//     PlcTask Inputs/GVL_iXlinker.EtherCAT_Master_ERxxxx.Beckhoff_ER3xxx.Beckhoff_ER3xxxEK1122.A_0012_ER3314_0002_0021.TC_Inputs_Channel_1.Status/Underrange <-> TC Inputs Channel 1/Status/Underrange
//     PlcTask Inputs/GVL_iXlinker.EtherCAT_Master_ERxxxx.Beckhoff_ER3xxx.Beckhoff_ER3xxxEK1122.A_0012_ER3314_0002_0021.TC_Inputs_Channel_2.Status/Underrange <-> TC Inputs Channel 2/Status/Underrange
//     PlcTask Inputs/GVL_iXlinker.EtherCAT_Master_ERxxxx.Beckhoff_ER3xxx.Beckhoff_ER3xxxEK1122.A_0012_ER3314_0002_0021.TC_Inputs_Channel_3.Status/Underrange <-> TC Inputs Channel 3/Status/Underrange
//     PlcTask Inputs/GVL_iXlinker.EtherCAT_Master_ERxxxx.Beckhoff_ER3xxx.Beckhoff_ER3xxxEK1122.A_0012_ER3314_0002_0021.TC_Inputs_Channel_4.Status/Underrange <-> TC Inputs Channel 4/Status/Underrange
//     PlcTask Inputs/GVL_iXlinker.EtherCAT_Master_ERxxxx.Beckhoff_ER3xxx.Beckhoff_ER3xxxEK1122.A_0012_ER3314_0002_0021.TC_Inputs_Channel_1.Status/Overrange <-> TC Inputs Channel 1/Status/Overrange
//     PlcTask Inputs/GVL_iXlinker.EtherCAT_Master_ERxxxx.Beckhoff_ER3xxx.Beckhoff_ER3xxxEK1122.A_0012_ER3314_0002_0021.TC_Inputs_Channel_2.Status/Overrange <-> TC Inputs Channel 2/Status/Overrange
//     PlcTask Inputs/GVL_iXlinker.EtherCAT_Master_ERxxxx.Beckhoff_ER3xxx.Beckhoff_ER3xxxEK1122.A_0012_ER3314_0002_0021.TC_Inputs_Channel_3.Status/Overrange <-> TC Inputs Channel 3/Status/Overrange
//     PlcTask Inputs/GVL_iXlinker.EtherCAT_Master_ERxxxx.Beckhoff_ER3xxx.Beckhoff_ER3xxxEK1122.A_0012_ER3314_0002_0021.TC_Inputs_Channel_4.Status/Overrange <-> TC Inputs Channel 4/Status/Overrange
//     PlcTask Inputs/GVL_iXlinker.EtherCAT_Master_ERxxxx.Beckhoff_ER3xxx.Beckhoff_ER3xxxEK1122.A_0012_ER3314_0002_0021.TC_Inputs_Channel_1.Status/Limit_1 <-> TC Inputs Channel 1/Status/Limit 1
//     PlcTask Inputs/GVL_iXlinker.EtherCAT_Master_ERxxxx.Beckhoff_ER3xxx.Beckhoff_ER3xxxEK1122.A_0012_ER3314_0002_0021.TC_Inputs_Channel_1.Status/Limit_2 <-> TC Inputs Channel 1/Status/Limit 2
//     PlcTask Inputs/GVL_iXlinker.EtherCAT_Master_ERxxxx.Beckhoff_ER3xxx.Beckhoff_ER3xxxEK1122.A_0012_ER3314_0002_0021.TC_Inputs_Channel_2.Status/Limit_1 <-> TC Inputs Channel 2/Status/Limit 1
//     PlcTask Inputs/GVL_iXlinker.EtherCAT_Master_ERxxxx.Beckhoff_ER3xxx.Beckhoff_ER3xxxEK1122.A_0012_ER3314_0002_0021.TC_Inputs_Channel_2.Status/Limit_2 <-> TC Inputs Channel 2/Status/Limit 2
//     PlcTask Inputs/GVL_iXlinker.EtherCAT_Master_ERxxxx.Beckhoff_ER3xxx.Beckhoff_ER3xxxEK1122.A_0012_ER3314_0002_0021.TC_Inputs_Channel_3.Status/Limit_1 <-> TC Inputs Channel 3/Status/Limit 1
//     PlcTask Inputs/GVL_iXlinker.EtherCAT_Master_ERxxxx.Beckhoff_ER3xxx.Beckhoff_ER3xxxEK1122.A_0012_ER3314_0002_0021.TC_Inputs_Channel_3.Status/Limit_2 <-> TC Inputs Channel 3/Status/Limit 2
//     PlcTask Inputs/GVL_iXlinker.EtherCAT_Master_ERxxxx.Beckhoff_ER3xxx.Beckhoff_ER3xxxEK1122.A_0012_ER3314_0002_0021.TC_Inputs_Channel_4.Status/Limit_1 <-> TC Inputs Channel 4/Status/Limit 1
//     PlcTask Inputs/GVL_iXlinker.EtherCAT_Master_ERxxxx.Beckhoff_ER3xxx.Beckhoff_ER3xxxEK1122.A_0012_ER3314_0002_0021.TC_Inputs_Channel_4.Status/Limit_2 <-> TC Inputs Channel 4/Status/Limit 2
//     PlcTask Inputs/GVL_iXlinker.EtherCAT_Master_ERxxxx.Beckhoff_ER3xxx.Beckhoff_ER3xxxEK1122.A_0012_ER3314_0002_0021.TC_Inputs_Channel_1.Status/Error <-> TC Inputs Channel 1/Status/Error
//     PlcTask Inputs/GVL_iXlinker.EtherCAT_Master_ERxxxx.Beckhoff_ER3xxx.Beckhoff_ER3xxxEK1122.A_0012_ER3314_0002_0021.TC_Inputs_Channel_2.Status/Error <-> TC Inputs Channel 2/Status/Error
//     PlcTask Inputs/GVL_iXlinker.EtherCAT_Master_ERxxxx.Beckhoff_ER3xxx.Beckhoff_ER3xxxEK1122.A_0012_ER3314_0002_0021.TC_Inputs_Channel_3.Status/Error <-> TC Inputs Channel 3/Status/Error
//     PlcTask Inputs/GVL_iXlinker.EtherCAT_Master_ERxxxx.Beckhoff_ER3xxx.Beckhoff_ER3xxxEK1122.A_0012_ER3314_0002_0021.TC_Inputs_Channel_4.Status/Error <-> TC Inputs Channel 4/Status/Error
//     PlcTask Inputs/GVL_iXlinker.EtherCAT_Master_ERxxxx.Beckhoff_ER3xxx.Beckhoff_ER3xxxEK1122.A_0012_ER3314_0002_0021.TC_Inputs_Channel_1.Status/TxPDO_State <-> TC Inputs Channel 1/Status/TxPDO State
//     PlcTask Inputs/GVL_iXlinker.EtherCAT_Master_ERxxxx.Beckhoff_ER3xxx.Beckhoff_ER3xxxEK1122.A_0012_ER3314_0002_0021.TC_Inputs_Channel_2.Status/TxPDO_State <-> TC Inputs Channel 2/Status/TxPDO State
//     PlcTask Inputs/GVL_iXlinker.EtherCAT_Master_ERxxxx.Beckhoff_ER3xxx.Beckhoff_ER3xxxEK1122.A_0012_ER3314_0002_0021.TC_Inputs_Channel_3.Status/TxPDO_State <-> TC Inputs Channel 3/Status/TxPDO State
//     PlcTask Inputs/GVL_iXlinker.EtherCAT_Master_ERxxxx.Beckhoff_ER3xxx.Beckhoff_ER3xxxEK1122.A_0012_ER3314_0002_0021.TC_Inputs_Channel_4.Status/TxPDO_State <-> TC Inputs Channel 4/Status/TxPDO State
//     PlcTask Inputs/GVL_iXlinker.EtherCAT_Master_ERxxxx.Beckhoff_ER3xxx.Beckhoff_ER3xxxEK1122.A_0012_ER3314_0002_0021.TC_Inputs_Channel_1.Status/TxPDO_Toggle <-> TC Inputs Channel 1/Status/TxPDO Toggle
//     PlcTask Inputs/GVL_iXlinker.EtherCAT_Master_ERxxxx.Beckhoff_ER3xxx.Beckhoff_ER3xxxEK1122.A_0012_ER3314_0002_0021.TC_Inputs_Channel_2.Status/TxPDO_Toggle <-> TC Inputs Channel 2/Status/TxPDO Toggle
//     PlcTask Inputs/GVL_iXlinker.EtherCAT_Master_ERxxxx.Beckhoff_ER3xxx.Beckhoff_ER3xxxEK1122.A_0012_ER3314_0002_0021.TC_Inputs_Channel_3.Status/TxPDO_Toggle <-> TC Inputs Channel 3/Status/TxPDO Toggle
//     PlcTask Inputs/GVL_iXlinker.EtherCAT_Master_ERxxxx.Beckhoff_ER3xxx.Beckhoff_ER3xxxEK1122.A_0012_ER3314_0002_0021.TC_Inputs_Channel_4.Status/TxPDO_Toggle <-> TC Inputs Channel 4/Status/TxPDO Toggle
//     PlcTask Inputs/GVL_iXlinker.EtherCAT_Master_ERxxxx.Beckhoff_ER3xxx.Beckhoff_ER3xxxEK1122.A_0012_ER3314_0002_0021.TC_Inputs_Channel_1.Value <-> TC Inputs Channel 1/Value
//     PlcTask Inputs/GVL_iXlinker.EtherCAT_Master_ERxxxx.Beckhoff_ER3xxx.Beckhoff_ER3xxxEK1122.A_0012_ER3314_0002_0021.TC_Inputs_Channel_2.Value <-> TC Inputs Channel 2/Value
//     PlcTask Inputs/GVL_iXlinker.EtherCAT_Master_ERxxxx.Beckhoff_ER3xxx.Beckhoff_ER3xxxEK1122.A_0012_ER3314_0002_0021.TC_Inputs_Channel_3.Value <-> TC Inputs Channel 3/Value
//     PlcTask Inputs/GVL_iXlinker.EtherCAT_Master_ERxxxx.Beckhoff_ER3xxx.Beckhoff_ER3xxxEK1122.A_0012_ER3314_0002_0021.TC_Inputs_Channel_4.Value <-> TC Inputs Channel 4/Value
//     PlcTask Inputs/GVL_iXlinker.EtherCAT_Master_ERxxxx.Beckhoff_ER3xxx.Beckhoff_ER3xxxEK1122.A_0012_ER3314_0002_0021.WcState.WcState <-> WcState/WcState
//     PlcTask Inputs/GVL_iXlinker.EtherCAT_Master_ERxxxx.Beckhoff_ER3xxx.Beckhoff_ER3xxxEK1122.A_0012_ER3314_0002_0021.WcState.InputToggle <-> WcState/InputToggle
//     PlcTask Inputs/GVL_iXlinker.EtherCAT_Master_ERxxxx.Beckhoff_ER3xxx.Beckhoff_ER3xxxEK1122.A_0012_ER3314_0002_0021.InfoData.AdsAddr <-> InfoData/AdsAddr
//     PlcTask Inputs/GVL_iXlinker.EtherCAT_Master_ERxxxx.Beckhoff_ER3xxx.Beckhoff_ER3xxxEK1122.A_0012_ER3314_0002_0021.InfoData.State <-> InfoData/State
//   PLC/PLC Instance <-> EtherCAT Master ERxxxx/Beckhoff ER4xxx
//     PlcTask Inputs/GVL_iXlinker.EtherCAT_Master_ERxxxx.Beckhoff_ER4xxx.InfoData.State <-> InfoData/State
//   PLC/PLC Instance <-> EtherCAT Master ERxxxx/Beckhoff ER4xxx/Beckhoff ER4xxxEK1122
//     PlcTask Inputs/GVL_iXlinker.EtherCAT_Master_ERxxxx.Beckhoff_ER4xxx.Beckhoff_ER4xxxEK1122.InfoData.State <-> InfoData/State
//   PLC/PLC Instance <-> EtherCAT Master ERxxxx/Beckhoff ER4xxx/Beckhoff ER4xxxEK1122/Beckhoff ER4xxxsub EK1100
//     PlcTask Inputs/GVL_iXlinker.EtherCAT_Master_ERxxxx.Beckhoff_ER4xxx.Beckhoff_ER4xxxEK1122.Beckhoff_ER4xxxsub_EK1100.InfoData.State <-> InfoData/State
//   PLC/PLC Instance <-> EtherCAT Master ERxxxx/Beckhoff ER4xxx/Beckhoff ER4xxxEK1122/A_0001(ER4174-0002-0016)
//     PlcTask Outputs/GVL_iXlinker.EtherCAT_Master_ERxxxx.Beckhoff_ER4xxx.Beckhoff_ER4xxxEK1122.A_0001_ER4174_0002_0016.AO_Outputs_Channel_1.Analog_output <-> AO Outputs Channel 1/Analog output
//     PlcTask Outputs/GVL_iXlinker.EtherCAT_Master_ERxxxx.Beckhoff_ER4xxx.Beckhoff_ER4xxxEK1122.A_0001_ER4174_0002_0016.AO_Outputs_Channel_2.Analog_output <-> AO Outputs Channel 2/Analog output
//     PlcTask Outputs/GVL_iXlinker.EtherCAT_Master_ERxxxx.Beckhoff_ER4xxx.Beckhoff_ER4xxxEK1122.A_0001_ER4174_0002_0016.AO_Outputs_Channel_3.Analog_output <-> AO Outputs Channel 3/Analog output
//     PlcTask Outputs/GVL_iXlinker.EtherCAT_Master_ERxxxx.Beckhoff_ER4xxx.Beckhoff_ER4xxxEK1122.A_0001_ER4174_0002_0016.AO_Outputs_Channel_4.Analog_output <-> AO Outputs Channel 4/Analog output
//     PlcTask Inputs/GVL_iXlinker.EtherCAT_Master_ERxxxx.Beckhoff_ER4xxx.Beckhoff_ER4xxxEK1122.A_0001_ER4174_0002_0016.WcState.WcState <-> WcState/WcState
//     PlcTask Inputs/GVL_iXlinker.EtherCAT_Master_ERxxxx.Beckhoff_ER4xxx.Beckhoff_ER4xxxEK1122.A_0001_ER4174_0002_0016.InfoData.AdsAddr <-> InfoData/AdsAddr
//     PlcTask Inputs/GVL_iXlinker.EtherCAT_Master_ERxxxx.Beckhoff_ER4xxx.Beckhoff_ER4xxxEK1122.A_0001_ER4174_0002_0016.InfoData.State <-> InfoData/State
//   PLC/PLC Instance <-> EtherCAT Master ERxxxx/Beckhoff ER4xxx/Beckhoff ER4xxxEK1122/A_0002(ER4174-0002-0019)
//     PlcTask Outputs/GVL_iXlinker.EtherCAT_Master_ERxxxx.Beckhoff_ER4xxx.Beckhoff_ER4xxxEK1122.A_0002_ER4174_0002_0019.AO_Outputs_Channel_1.Analog_output <-> AO Outputs Channel 1/Analog output
//     PlcTask Outputs/GVL_iXlinker.EtherCAT_Master_ERxxxx.Beckhoff_ER4xxx.Beckhoff_ER4xxxEK1122.A_0002_ER4174_0002_0019.AO_Outputs_Channel_2.Analog_output <-> AO Outputs Channel 2/Analog output
//     PlcTask Outputs/GVL_iXlinker.EtherCAT_Master_ERxxxx.Beckhoff_ER4xxx.Beckhoff_ER4xxxEK1122.A_0002_ER4174_0002_0019.AO_Outputs_Channel_3.Analog_output <-> AO Outputs Channel 3/Analog output
//     PlcTask Outputs/GVL_iXlinker.EtherCAT_Master_ERxxxx.Beckhoff_ER4xxx.Beckhoff_ER4xxxEK1122.A_0002_ER4174_0002_0019.AO_Outputs_Channel_4.Analog_output <-> AO Outputs Channel 4/Analog output
//     PlcTask Inputs/GVL_iXlinker.EtherCAT_Master_ERxxxx.Beckhoff_ER4xxx.Beckhoff_ER4xxxEK1122.A_0002_ER4174_0002_0019.WcState.WcState <-> WcState/WcState
//     PlcTask Inputs/GVL_iXlinker.EtherCAT_Master_ERxxxx.Beckhoff_ER4xxx.Beckhoff_ER4xxxEK1122.A_0002_ER4174_0002_0019.InfoData.AdsAddr <-> InfoData/AdsAddr
//     PlcTask Inputs/GVL_iXlinker.EtherCAT_Master_ERxxxx.Beckhoff_ER4xxx.Beckhoff_ER4xxxEK1122.A_0002_ER4174_0002_0019.InfoData.State <-> InfoData/State
//   PLC/PLC Instance <-> EtherCAT Master ERxxxx/Beckhoff ER4xxx/Beckhoff ER4xxxEK1122/A_0003(ER4374-0002-0018)
//     PlcTask Inputs/GVL_iXlinker.EtherCAT_Master_ERxxxx.Beckhoff_ER4xxx.Beckhoff_ER4xxxEK1122.A_0003_ER4374_0002_0018.AI_Inputs_Channel_1.Status/Underrange <-> AI Inputs Channel 1/Status/Underrange
//     PlcTask Inputs/GVL_iXlinker.EtherCAT_Master_ERxxxx.Beckhoff_ER4xxx.Beckhoff_ER4xxxEK1122.A_0003_ER4374_0002_0018.AI_Inputs_Channel_2.Status/Underrange <-> AI Inputs Channel 2/Status/Underrange
//     PlcTask Inputs/GVL_iXlinker.EtherCAT_Master_ERxxxx.Beckhoff_ER4xxx.Beckhoff_ER4xxxEK1122.A_0003_ER4374_0002_0018.AI_Inputs_Channel_1.Status/Overrange <-> AI Inputs Channel 1/Status/Overrange
//     PlcTask Inputs/GVL_iXlinker.EtherCAT_Master_ERxxxx.Beckhoff_ER4xxx.Beckhoff_ER4xxxEK1122.A_0003_ER4374_0002_0018.AI_Inputs_Channel_2.Status/Overrange <-> AI Inputs Channel 2/Status/Overrange
//     PlcTask Inputs/GVL_iXlinker.EtherCAT_Master_ERxxxx.Beckhoff_ER4xxx.Beckhoff_ER4xxxEK1122.A_0003_ER4374_0002_0018.AI_Inputs_Channel_1.Status/Limit_1 <-> AI Inputs Channel 1/Status/Limit 1
//     PlcTask Inputs/GVL_iXlinker.EtherCAT_Master_ERxxxx.Beckhoff_ER4xxx.Beckhoff_ER4xxxEK1122.A_0003_ER4374_0002_0018.AI_Inputs_Channel_1.Status/Limit_2 <-> AI Inputs Channel 1/Status/Limit 2
//     PlcTask Inputs/GVL_iXlinker.EtherCAT_Master_ERxxxx.Beckhoff_ER4xxx.Beckhoff_ER4xxxEK1122.A_0003_ER4374_0002_0018.AI_Inputs_Channel_2.Status/Limit_1 <-> AI Inputs Channel 2/Status/Limit 1
//     PlcTask Inputs/GVL_iXlinker.EtherCAT_Master_ERxxxx.Beckhoff_ER4xxx.Beckhoff_ER4xxxEK1122.A_0003_ER4374_0002_0018.AI_Inputs_Channel_2.Status/Limit_2 <-> AI Inputs Channel 2/Status/Limit 2
//     PlcTask Inputs/GVL_iXlinker.EtherCAT_Master_ERxxxx.Beckhoff_ER4xxx.Beckhoff_ER4xxxEK1122.A_0003_ER4374_0002_0018.AI_Inputs_Channel_1.Status/Error <-> AI Inputs Channel 1/Status/Error
//     PlcTask Inputs/GVL_iXlinker.EtherCAT_Master_ERxxxx.Beckhoff_ER4xxx.Beckhoff_ER4xxxEK1122.A_0003_ER4374_0002_0018.AI_Inputs_Channel_2.Status/Error <-> AI Inputs Channel 2/Status/Error
//     PlcTask Inputs/GVL_iXlinker.EtherCAT_Master_ERxxxx.Beckhoff_ER4xxx.Beckhoff_ER4xxxEK1122.A_0003_ER4374_0002_0018.AI_Inputs_Channel_1.Status/Sync_error <-> AI Inputs Channel 1/Status/Sync error
//     PlcTask Inputs/GVL_iXlinker.EtherCAT_Master_ERxxxx.Beckhoff_ER4xxx.Beckhoff_ER4xxxEK1122.A_0003_ER4374_0002_0018.AI_Inputs_Channel_2.Status/Sync_error <-> AI Inputs Channel 2/Status/Sync error
//     PlcTask Inputs/GVL_iXlinker.EtherCAT_Master_ERxxxx.Beckhoff_ER4xxx.Beckhoff_ER4xxxEK1122.A_0003_ER4374_0002_0018.AI_Inputs_Channel_1.Status/TxPDO_State <-> AI Inputs Channel 1/Status/TxPDO State
//     PlcTask Inputs/GVL_iXlinker.EtherCAT_Master_ERxxxx.Beckhoff_ER4xxx.Beckhoff_ER4xxxEK1122.A_0003_ER4374_0002_0018.AI_Inputs_Channel_2.Status/TxPDO_State <-> AI Inputs Channel 2/Status/TxPDO State
//     PlcTask Inputs/GVL_iXlinker.EtherCAT_Master_ERxxxx.Beckhoff_ER4xxx.Beckhoff_ER4xxxEK1122.A_0003_ER4374_0002_0018.AI_Inputs_Channel_1.Status/TxPDO_Toggle <-> AI Inputs Channel 1/Status/TxPDO Toggle
//     PlcTask Inputs/GVL_iXlinker.EtherCAT_Master_ERxxxx.Beckhoff_ER4xxx.Beckhoff_ER4xxxEK1122.A_0003_ER4374_0002_0018.AI_Inputs_Channel_2.Status/TxPDO_Toggle <-> AI Inputs Channel 2/Status/TxPDO Toggle
//     PlcTask Inputs/GVL_iXlinker.EtherCAT_Master_ERxxxx.Beckhoff_ER4xxx.Beckhoff_ER4xxxEK1122.A_0003_ER4374_0002_0018.AI_Inputs_Channel_1.Value <-> AI Inputs Channel 1/Value
//     PlcTask Inputs/GVL_iXlinker.EtherCAT_Master_ERxxxx.Beckhoff_ER4xxx.Beckhoff_ER4xxxEK1122.A_0003_ER4374_0002_0018.AI_Inputs_Channel_2.Value <-> AI Inputs Channel 2/Value
//     PlcTask Outputs/GVL_iXlinker.EtherCAT_Master_ERxxxx.Beckhoff_ER4xxx.Beckhoff_ER4xxxEK1122.A_0003_ER4374_0002_0018.AO_Outputs_Channel_3.Analog_output <-> AO Outputs Channel 3/Analog output
//     PlcTask Outputs/GVL_iXlinker.EtherCAT_Master_ERxxxx.Beckhoff_ER4xxx.Beckhoff_ER4xxxEK1122.A_0003_ER4374_0002_0018.AO_Outputs_Channel_4.Analog_output <-> AO Outputs Channel 4/Analog output
//     PlcTask Inputs/GVL_iXlinker.EtherCAT_Master_ERxxxx.Beckhoff_ER4xxx.Beckhoff_ER4xxxEK1122.A_0003_ER4374_0002_0018.WcState.WcState <-> WcState/WcState
//     PlcTask Inputs/GVL_iXlinker.EtherCAT_Master_ERxxxx.Beckhoff_ER4xxx.Beckhoff_ER4xxxEK1122.A_0003_ER4374_0002_0018.WcState.InputToggle <-> WcState/InputToggle
//     PlcTask Inputs/GVL_iXlinker.EtherCAT_Master_ERxxxx.Beckhoff_ER4xxx.Beckhoff_ER4xxxEK1122.A_0003_ER4374_0002_0018.InfoData.AdsAddr <-> InfoData/AdsAddr
//     PlcTask Inputs/GVL_iXlinker.EtherCAT_Master_ERxxxx.Beckhoff_ER4xxx.Beckhoff_ER4xxxEK1122.A_0003_ER4374_0002_0018.InfoData.State <-> InfoData/State
//   PLC/PLC Instance <-> EtherCAT Master ERxxxx/Beckhoff ER4xxx/Beckhoff ER4xxxEK1122/A_0004(ER4374-0002-0019)
//     PlcTask Inputs/GVL_iXlinker.EtherCAT_Master_ERxxxx.Beckhoff_ER4xxx.Beckhoff_ER4xxxEK1122.A_0004_ER4374_0002_0019.AI_Inputs_Channel_1.Status/Underrange <-> AI Inputs Channel 1/Status/Underrange
//     PlcTask Inputs/GVL_iXlinker.EtherCAT_Master_ERxxxx.Beckhoff_ER4xxx.Beckhoff_ER4xxxEK1122.A_0004_ER4374_0002_0019.AI_Inputs_Channel_2.Status/Underrange <-> AI Inputs Channel 2/Status/Underrange
//     PlcTask Inputs/GVL_iXlinker.EtherCAT_Master_ERxxxx.Beckhoff_ER4xxx.Beckhoff_ER4xxxEK1122.A_0004_ER4374_0002_0019.AI_Inputs_Channel_1.Status/Overrange <-> AI Inputs Channel 1/Status/Overrange
//     PlcTask Inputs/GVL_iXlinker.EtherCAT_Master_ERxxxx.Beckhoff_ER4xxx.Beckhoff_ER4xxxEK1122.A_0004_ER4374_0002_0019.AI_Inputs_Channel_2.Status/Overrange <-> AI Inputs Channel 2/Status/Overrange
//     PlcTask Inputs/GVL_iXlinker.EtherCAT_Master_ERxxxx.Beckhoff_ER4xxx.Beckhoff_ER4xxxEK1122.A_0004_ER4374_0002_0019.AI_Inputs_Channel_1.Status/Limit_1 <-> AI Inputs Channel 1/Status/Limit 1
//     PlcTask Inputs/GVL_iXlinker.EtherCAT_Master_ERxxxx.Beckhoff_ER4xxx.Beckhoff_ER4xxxEK1122.A_0004_ER4374_0002_0019.AI_Inputs_Channel_1.Status/Limit_2 <-> AI Inputs Channel 1/Status/Limit 2
//     PlcTask Inputs/GVL_iXlinker.EtherCAT_Master_ERxxxx.Beckhoff_ER4xxx.Beckhoff_ER4xxxEK1122.A_0004_ER4374_0002_0019.AI_Inputs_Channel_2.Status/Limit_1 <-> AI Inputs Channel 2/Status/Limit 1
//     PlcTask Inputs/GVL_iXlinker.EtherCAT_Master_ERxxxx.Beckhoff_ER4xxx.Beckhoff_ER4xxxEK1122.A_0004_ER4374_0002_0019.AI_Inputs_Channel_2.Status/Limit_2 <-> AI Inputs Channel 2/Status/Limit 2
//     PlcTask Inputs/GVL_iXlinker.EtherCAT_Master_ERxxxx.Beckhoff_ER4xxx.Beckhoff_ER4xxxEK1122.A_0004_ER4374_0002_0019.AI_Inputs_Channel_1.Status/Error <-> AI Inputs Channel 1/Status/Error
//     PlcTask Inputs/GVL_iXlinker.EtherCAT_Master_ERxxxx.Beckhoff_ER4xxx.Beckhoff_ER4xxxEK1122.A_0004_ER4374_0002_0019.AI_Inputs_Channel_2.Status/Error <-> AI Inputs Channel 2/Status/Error
//     PlcTask Inputs/GVL_iXlinker.EtherCAT_Master_ERxxxx.Beckhoff_ER4xxx.Beckhoff_ER4xxxEK1122.A_0004_ER4374_0002_0019.AI_Inputs_Channel_1.Status/Sync_error <-> AI Inputs Channel 1/Status/Sync error
//     PlcTask Inputs/GVL_iXlinker.EtherCAT_Master_ERxxxx.Beckhoff_ER4xxx.Beckhoff_ER4xxxEK1122.A_0004_ER4374_0002_0019.AI_Inputs_Channel_2.Status/Sync_error <-> AI Inputs Channel 2/Status/Sync error
//     PlcTask Inputs/GVL_iXlinker.EtherCAT_Master_ERxxxx.Beckhoff_ER4xxx.Beckhoff_ER4xxxEK1122.A_0004_ER4374_0002_0019.AI_Inputs_Channel_1.Status/TxPDO_State <-> AI Inputs Channel 1/Status/TxPDO State
//     PlcTask Inputs/GVL_iXlinker.EtherCAT_Master_ERxxxx.Beckhoff_ER4xxx.Beckhoff_ER4xxxEK1122.A_0004_ER4374_0002_0019.AI_Inputs_Channel_2.Status/TxPDO_State <-> AI Inputs Channel 2/Status/TxPDO State
//     PlcTask Inputs/GVL_iXlinker.EtherCAT_Master_ERxxxx.Beckhoff_ER4xxx.Beckhoff_ER4xxxEK1122.A_0004_ER4374_0002_0019.AI_Inputs_Channel_1.Status/TxPDO_Toggle <-> AI Inputs Channel 1/Status/TxPDO Toggle
//     PlcTask Inputs/GVL_iXlinker.EtherCAT_Master_ERxxxx.Beckhoff_ER4xxx.Beckhoff_ER4xxxEK1122.A_0004_ER4374_0002_0019.AI_Inputs_Channel_2.Status/TxPDO_Toggle <-> AI Inputs Channel 2/Status/TxPDO Toggle
//     PlcTask Inputs/GVL_iXlinker.EtherCAT_Master_ERxxxx.Beckhoff_ER4xxx.Beckhoff_ER4xxxEK1122.A_0004_ER4374_0002_0019.AI_Inputs_Channel_1.Value <-> AI Inputs Channel 1/Value
//     PlcTask Inputs/GVL_iXlinker.EtherCAT_Master_ERxxxx.Beckhoff_ER4xxx.Beckhoff_ER4xxxEK1122.A_0004_ER4374_0002_0019.AI_Inputs_Channel_2.Value <-> AI Inputs Channel 2/Value
//     PlcTask Outputs/GVL_iXlinker.EtherCAT_Master_ERxxxx.Beckhoff_ER4xxx.Beckhoff_ER4xxxEK1122.A_0004_ER4374_0002_0019.AO_Outputs_Channel_3.Analog_output <-> AO Outputs Channel 3/Analog output
//     PlcTask Outputs/GVL_iXlinker.EtherCAT_Master_ERxxxx.Beckhoff_ER4xxx.Beckhoff_ER4xxxEK1122.A_0004_ER4374_0002_0019.AO_Outputs_Channel_4.Analog_output <-> AO Outputs Channel 4/Analog output
//     PlcTask Inputs/GVL_iXlinker.EtherCAT_Master_ERxxxx.Beckhoff_ER4xxx.Beckhoff_ER4xxxEK1122.A_0004_ER4374_0002_0019.WcState.WcState <-> WcState/WcState
//     PlcTask Inputs/GVL_iXlinker.EtherCAT_Master_ERxxxx.Beckhoff_ER4xxx.Beckhoff_ER4xxxEK1122.A_0004_ER4374_0002_0019.WcState.InputToggle <-> WcState/InputToggle
//     PlcTask Inputs/GVL_iXlinker.EtherCAT_Master_ERxxxx.Beckhoff_ER4xxx.Beckhoff_ER4xxxEK1122.A_0004_ER4374_0002_0019.InfoData.AdsAddr <-> InfoData/AdsAddr
//     PlcTask Inputs/GVL_iXlinker.EtherCAT_Master_ERxxxx.Beckhoff_ER4xxx.Beckhoff_ER4xxxEK1122.A_0004_ER4374_0002_0019.InfoData.State <-> InfoData/State
//   PLC/PLC Instance <-> EtherCAT Master ERxxxx/Beckhoff ER5xxx
//     PlcTask Inputs/GVL_iXlinker.EtherCAT_Master_ERxxxx.Beckhoff_ER5xxx.InfoData.State <-> InfoData/State
//   PLC/PLC Instance <-> EtherCAT Master ERxxxx/Beckhoff ER5xxx/Beckhoff ER5xxxEK1122
//     PlcTask Inputs/GVL_iXlinker.EtherCAT_Master_ERxxxx.Beckhoff_ER5xxx.Beckhoff_ER5xxxEK1122.InfoData.State <-> InfoData/State
//   PLC/PLC Instance <-> EtherCAT Master ERxxxx/Beckhoff ER5xxx/Beckhoff ER5xxxEK1122/Beckhoff ER5xxxsub EK1100
//     PlcTask Inputs/GVL_iXlinker.EtherCAT_Master_ERxxxx.Beckhoff_ER5xxx.Beckhoff_ER5xxxEK1122.Beckhoff_ER5xxxsub_EK1100.InfoData.State <-> InfoData/State
//   PLC/PLC Instance <-> EtherCAT Master ERxxxx/Beckhoff ER5xxx/Beckhoff ER5xxxEK1122/A_0001(ER5101-0002-0019)
//     PlcTask Inputs/GVL_iXlinker.EtherCAT_Master_ERxxxx.Beckhoff_ER5xxx.Beckhoff_ER5xxxEK1122.A_0001_ER5101_0002_0019.ENC_Status_compact.Status/Latch_C_valid <-> ENC Status compact/Status/Latch C valid
//     PlcTask Inputs/GVL_iXlinker.EtherCAT_Master_ERxxxx.Beckhoff_ER5xxx.Beckhoff_ER5xxxEK1122.A_0001_ER5101_0002_0019.ENC_Status_compact.Status/Set_counter_done <-> ENC Status compact/Status/Set counter done
//     PlcTask Inputs/GVL_iXlinker.EtherCAT_Master_ERxxxx.Beckhoff_ER5xxx.Beckhoff_ER5xxxEK1122.A_0001_ER5101_0002_0019.ENC_Status_compact.Status/Counter_underflow <-> ENC Status compact/Status/Counter underflow
//     PlcTask Inputs/GVL_iXlinker.EtherCAT_Master_ERxxxx.Beckhoff_ER5xxx.Beckhoff_ER5xxxEK1122.A_0001_ER5101_0002_0019.ENC_Status_compact.Status/Counter_overflow <-> ENC Status compact/Status/Counter overflow
//     PlcTask Inputs/GVL_iXlinker.EtherCAT_Master_ERxxxx.Beckhoff_ER5xxx.Beckhoff_ER5xxxEK1122.A_0001_ER5101_0002_0019.ENC_Status_compact.Status/Open_circuit <-> ENC Status compact/Status/Open circuit
//     PlcTask Inputs/GVL_iXlinker.EtherCAT_Master_ERxxxx.Beckhoff_ER5xxx.Beckhoff_ER5xxxEK1122.A_0001_ER5101_0002_0019.ENC_Status_compact.Status/Extrapolation_stall <-> ENC Status compact/Status/Extrapolation stall
//     PlcTask Inputs/GVL_iXlinker.EtherCAT_Master_ERxxxx.Beckhoff_ER5xxx.Beckhoff_ER5xxxEK1122.A_0001_ER5101_0002_0019.ENC_Status_compact.Status/Status_of_input_A <-> ENC Status compact/Status/Status of input A
//     PlcTask Inputs/GVL_iXlinker.EtherCAT_Master_ERxxxx.Beckhoff_ER5xxx.Beckhoff_ER5xxxEK1122.A_0001_ER5101_0002_0019.ENC_Status_compact.Status/Status_of_input_B <-> ENC Status compact/Status/Status of input B
//     PlcTask Inputs/GVL_iXlinker.EtherCAT_Master_ERxxxx.Beckhoff_ER5xxx.Beckhoff_ER5xxxEK1122.A_0001_ER5101_0002_0019.ENC_Status_compact.Status/Status_of_input_C <-> ENC Status compact/Status/Status of input C
//     PlcTask Inputs/GVL_iXlinker.EtherCAT_Master_ERxxxx.Beckhoff_ER5xxx.Beckhoff_ER5xxxEK1122.A_0001_ER5101_0002_0019.ENC_Status_compact.Status/Sync_error <-> ENC Status compact/Status/Sync error
//     PlcTask Inputs/GVL_iXlinker.EtherCAT_Master_ERxxxx.Beckhoff_ER5xxx.Beckhoff_ER5xxxEK1122.A_0001_ER5101_0002_0019.ENC_Status_compact.Status/TxPDO_State <-> ENC Status compact/Status/TxPDO State
//     PlcTask Inputs/GVL_iXlinker.EtherCAT_Master_ERxxxx.Beckhoff_ER5xxx.Beckhoff_ER5xxxEK1122.A_0001_ER5101_0002_0019.ENC_Status_compact.Status/TxPDO_Toggle <-> ENC Status compact/Status/TxPDO Toggle
//     PlcTask Inputs/GVL_iXlinker.EtherCAT_Master_ERxxxx.Beckhoff_ER5xxx.Beckhoff_ER5xxxEK1122.A_0001_ER5101_0002_0019.ENC_Status_compact.Counter_value <-> ENC Status compact/Counter value
//     PlcTask Inputs/GVL_iXlinker.EtherCAT_Master_ERxxxx.Beckhoff_ER5xxx.Beckhoff_ER5xxxEK1122.A_0001_ER5101_0002_0019.ENC_Status_compact.Latch_value <-> ENC Status compact/Latch value
//     PlcTask Outputs/GVL_iXlinker.EtherCAT_Master_ERxxxx.Beckhoff_ER5xxx.Beckhoff_ER5xxxEK1122.A_0001_ER5101_0002_0019.ENC_Control_compact.Control/Enable_latch_C <-> ENC Control compact/Control/Enable latch C
//     PlcTask Outputs/GVL_iXlinker.EtherCAT_Master_ERxxxx.Beckhoff_ER5xxx.Beckhoff_ER5xxxEK1122.A_0001_ER5101_0002_0019.ENC_Control_compact.Control/Set_counter <-> ENC Control compact/Control/Set counter
//     PlcTask Outputs/GVL_iXlinker.EtherCAT_Master_ERxxxx.Beckhoff_ER5xxx.Beckhoff_ER5xxxEK1122.A_0001_ER5101_0002_0019.ENC_Control_compact.Set_counter_value <-> ENC Control compact/Set counter value
//     PlcTask Inputs/GVL_iXlinker.EtherCAT_Master_ERxxxx.Beckhoff_ER5xxx.Beckhoff_ER5xxxEK1122.A_0001_ER5101_0002_0019.WcState.WcState <-> WcState/WcState
//     PlcTask Inputs/GVL_iXlinker.EtherCAT_Master_ERxxxx.Beckhoff_ER5xxx.Beckhoff_ER5xxxEK1122.A_0001_ER5101_0002_0019.WcState.InputToggle <-> WcState/InputToggle
//     PlcTask Inputs/GVL_iXlinker.EtherCAT_Master_ERxxxx.Beckhoff_ER5xxx.Beckhoff_ER5xxxEK1122.A_0001_ER5101_0002_0019.InfoData.AdsAddr <-> InfoData/AdsAddr
//     PlcTask Inputs/GVL_iXlinker.EtherCAT_Master_ERxxxx.Beckhoff_ER5xxx.Beckhoff_ER5xxxEK1122.A_0001_ER5101_0002_0019.InfoData.State <-> InfoData/State
//   PLC/PLC Instance <-> EtherCAT Master ERxxxx/Beckhoff ER5xxx/Beckhoff ER5xxxEK1122/A_0002(ER5101-1002-0017)
//     PlcTask Inputs/GVL_iXlinker.EtherCAT_Master_ERxxxx.Beckhoff_ER5xxx.Beckhoff_ER5xxxEK1122.A_0002_ER5101_1002_0017.ENC_Status_compact.Status/Latch_C_valid <-> ENC Status compact/Status/Latch C valid
//     PlcTask Inputs/GVL_iXlinker.EtherCAT_Master_ERxxxx.Beckhoff_ER5xxx.Beckhoff_ER5xxxEK1122.A_0002_ER5101_1002_0017.ENC_Status_compact.Status/Set_counter_done <-> ENC Status compact/Status/Set counter done
//     PlcTask Inputs/GVL_iXlinker.EtherCAT_Master_ERxxxx.Beckhoff_ER5xxx.Beckhoff_ER5xxxEK1122.A_0002_ER5101_1002_0017.ENC_Status_compact.Status/Counter_underflow <-> ENC Status compact/Status/Counter underflow
//     PlcTask Inputs/GVL_iXlinker.EtherCAT_Master_ERxxxx.Beckhoff_ER5xxx.Beckhoff_ER5xxxEK1122.A_0002_ER5101_1002_0017.ENC_Status_compact.Status/Counter_overflow <-> ENC Status compact/Status/Counter overflow
//     PlcTask Inputs/GVL_iXlinker.EtherCAT_Master_ERxxxx.Beckhoff_ER5xxx.Beckhoff_ER5xxxEK1122.A_0002_ER5101_1002_0017.ENC_Status_compact.Status/Open_circuit <-> ENC Status compact/Status/Open circuit
//     PlcTask Inputs/GVL_iXlinker.EtherCAT_Master_ERxxxx.Beckhoff_ER5xxx.Beckhoff_ER5xxxEK1122.A_0002_ER5101_1002_0017.ENC_Status_compact.Status/Extrapolation_stall <-> ENC Status compact/Status/Extrapolation stall
//     PlcTask Inputs/GVL_iXlinker.EtherCAT_Master_ERxxxx.Beckhoff_ER5xxx.Beckhoff_ER5xxxEK1122.A_0002_ER5101_1002_0017.ENC_Status_compact.Status/Status_of_input_A <-> ENC Status compact/Status/Status of input A
//     PlcTask Inputs/GVL_iXlinker.EtherCAT_Master_ERxxxx.Beckhoff_ER5xxx.Beckhoff_ER5xxxEK1122.A_0002_ER5101_1002_0017.ENC_Status_compact.Status/Status_of_input_B <-> ENC Status compact/Status/Status of input B
//     PlcTask Inputs/GVL_iXlinker.EtherCAT_Master_ERxxxx.Beckhoff_ER5xxx.Beckhoff_ER5xxxEK1122.A_0002_ER5101_1002_0017.ENC_Status_compact.Status/Status_of_input_C <-> ENC Status compact/Status/Status of input C
//     PlcTask Inputs/GVL_iXlinker.EtherCAT_Master_ERxxxx.Beckhoff_ER5xxx.Beckhoff_ER5xxxEK1122.A_0002_ER5101_1002_0017.ENC_Status_compact.Status/Sync_error <-> ENC Status compact/Status/Sync error
//     PlcTask Inputs/GVL_iXlinker.EtherCAT_Master_ERxxxx.Beckhoff_ER5xxx.Beckhoff_ER5xxxEK1122.A_0002_ER5101_1002_0017.ENC_Status_compact.Status/TxPDO_State <-> ENC Status compact/Status/TxPDO State
//     PlcTask Inputs/GVL_iXlinker.EtherCAT_Master_ERxxxx.Beckhoff_ER5xxx.Beckhoff_ER5xxxEK1122.A_0002_ER5101_1002_0017.ENC_Status_compact.Status/TxPDO_Toggle <-> ENC Status compact/Status/TxPDO Toggle
//     PlcTask Inputs/GVL_iXlinker.EtherCAT_Master_ERxxxx.Beckhoff_ER5xxx.Beckhoff_ER5xxxEK1122.A_0002_ER5101_1002_0017.ENC_Status_compact.Counter_value <-> ENC Status compact/Counter value
//     PlcTask Inputs/GVL_iXlinker.EtherCAT_Master_ERxxxx.Beckhoff_ER5xxx.Beckhoff_ER5xxxEK1122.A_0002_ER5101_1002_0017.ENC_Status_compact.Latch_value <-> ENC Status compact/Latch value
//     PlcTask Outputs/GVL_iXlinker.EtherCAT_Master_ERxxxx.Beckhoff_ER5xxx.Beckhoff_ER5xxxEK1122.A_0002_ER5101_1002_0017.ENC_Control_compact.Control/Enable_latch_C <-> ENC Control compact/Control/Enable latch C
//     PlcTask Outputs/GVL_iXlinker.EtherCAT_Master_ERxxxx.Beckhoff_ER5xxx.Beckhoff_ER5xxxEK1122.A_0002_ER5101_1002_0017.ENC_Control_compact.Control/Set_counter <-> ENC Control compact/Control/Set counter
//     PlcTask Outputs/GVL_iXlinker.EtherCAT_Master_ERxxxx.Beckhoff_ER5xxx.Beckhoff_ER5xxxEK1122.A_0002_ER5101_1002_0017.ENC_Control_compact.Set_counter_value <-> ENC Control compact/Set counter value
//     PlcTask Inputs/GVL_iXlinker.EtherCAT_Master_ERxxxx.Beckhoff_ER5xxx.Beckhoff_ER5xxxEK1122.A_0002_ER5101_1002_0017.WcState.WcState <-> WcState/WcState
//     PlcTask Inputs/GVL_iXlinker.EtherCAT_Master_ERxxxx.Beckhoff_ER5xxx.Beckhoff_ER5xxxEK1122.A_0002_ER5101_1002_0017.WcState.InputToggle <-> WcState/InputToggle
//     PlcTask Inputs/GVL_iXlinker.EtherCAT_Master_ERxxxx.Beckhoff_ER5xxx.Beckhoff_ER5xxxEK1122.A_0002_ER5101_1002_0017.InfoData.AdsAddr <-> InfoData/AdsAddr
//     PlcTask Inputs/GVL_iXlinker.EtherCAT_Master_ERxxxx.Beckhoff_ER5xxx.Beckhoff_ER5xxxEK1122.A_0002_ER5101_1002_0017.InfoData.State <-> InfoData/State
//   PLC/PLC Instance <-> EtherCAT Master ERxxxx/Beckhoff ER5xxx/Beckhoff ER5xxxEK1122/A_0003(ER5151-0002-0018)
//     PlcTask Inputs/GVL_iXlinker.EtherCAT_Master_ERxxxx.Beckhoff_ER5xxx.Beckhoff_ER5xxxEK1122.A_0003_ER5151_0002_0018.ENC_Status_compact.Status/Latch_C_valid <-> ENC Status compact/Status/Latch C valid
//     PlcTask Inputs/GVL_iXlinker.EtherCAT_Master_ERxxxx.Beckhoff_ER5xxx.Beckhoff_ER5xxxEK1122.A_0003_ER5151_0002_0018.ENC_Status_compact.Status/Latch_extern_valid <-> ENC Status compact/Status/Latch extern valid
//     PlcTask Inputs/GVL_iXlinker.EtherCAT_Master_ERxxxx.Beckhoff_ER5xxx.Beckhoff_ER5xxxEK1122.A_0003_ER5151_0002_0018.ENC_Status_compact.Status/Set_counter_done <-> ENC Status compact/Status/Set counter done
//     PlcTask Inputs/GVL_iXlinker.EtherCAT_Master_ERxxxx.Beckhoff_ER5xxx.Beckhoff_ER5xxxEK1122.A_0003_ER5151_0002_0018.ENC_Status_compact.Status/Counter_underflow <-> ENC Status compact/Status/Counter underflow
//     PlcTask Inputs/GVL_iXlinker.EtherCAT_Master_ERxxxx.Beckhoff_ER5xxx.Beckhoff_ER5xxxEK1122.A_0003_ER5151_0002_0018.ENC_Status_compact.Status/Counter_overflow <-> ENC Status compact/Status/Counter overflow
//     PlcTask Inputs/GVL_iXlinker.EtherCAT_Master_ERxxxx.Beckhoff_ER5xxx.Beckhoff_ER5xxxEK1122.A_0003_ER5151_0002_0018.ENC_Status_compact.Status/Status_of_input_status <-> ENC Status compact/Status/Status of input status
//     PlcTask Inputs/GVL_iXlinker.EtherCAT_Master_ERxxxx.Beckhoff_ER5xxx.Beckhoff_ER5xxxEK1122.A_0003_ER5151_0002_0018.ENC_Status_compact.Status/Open_circuit <-> ENC Status compact/Status/Open circuit
//     PlcTask Inputs/GVL_iXlinker.EtherCAT_Master_ERxxxx.Beckhoff_ER5xxx.Beckhoff_ER5xxxEK1122.A_0003_ER5151_0002_0018.ENC_Status_compact.Status/Extrapolation_stall <-> ENC Status compact/Status/Extrapolation stall
//     PlcTask Inputs/GVL_iXlinker.EtherCAT_Master_ERxxxx.Beckhoff_ER5xxx.Beckhoff_ER5xxxEK1122.A_0003_ER5151_0002_0018.ENC_Status_compact.Status/Status_of_input_A <-> ENC Status compact/Status/Status of input A
//     PlcTask Inputs/GVL_iXlinker.EtherCAT_Master_ERxxxx.Beckhoff_ER5xxx.Beckhoff_ER5xxxEK1122.A_0003_ER5151_0002_0018.ENC_Status_compact.Status/Status_of_input_B <-> ENC Status compact/Status/Status of input B
//     PlcTask Inputs/GVL_iXlinker.EtherCAT_Master_ERxxxx.Beckhoff_ER5xxx.Beckhoff_ER5xxxEK1122.A_0003_ER5151_0002_0018.ENC_Status_compact.Status/Status_of_input_C <-> ENC Status compact/Status/Status of input C
//     PlcTask Inputs/GVL_iXlinker.EtherCAT_Master_ERxxxx.Beckhoff_ER5xxx.Beckhoff_ER5xxxEK1122.A_0003_ER5151_0002_0018.ENC_Status_compact.Status/Status_of_input_gate <-> ENC Status compact/Status/Status of input gate
//     PlcTask Inputs/GVL_iXlinker.EtherCAT_Master_ERxxxx.Beckhoff_ER5xxx.Beckhoff_ER5xxxEK1122.A_0003_ER5151_0002_0018.ENC_Status_compact.Status/Status_of_extern_latch <-> ENC Status compact/Status/Status of extern latch
//     PlcTask Inputs/GVL_iXlinker.EtherCAT_Master_ERxxxx.Beckhoff_ER5xxx.Beckhoff_ER5xxxEK1122.A_0003_ER5151_0002_0018.ENC_Status_compact.Status/Sync_error <-> ENC Status compact/Status/Sync error
//     PlcTask Inputs/GVL_iXlinker.EtherCAT_Master_ERxxxx.Beckhoff_ER5xxx.Beckhoff_ER5xxxEK1122.A_0003_ER5151_0002_0018.ENC_Status_compact.Status/TxPDO_State <-> ENC Status compact/Status/TxPDO State
//     PlcTask Inputs/GVL_iXlinker.EtherCAT_Master_ERxxxx.Beckhoff_ER5xxx.Beckhoff_ER5xxxEK1122.A_0003_ER5151_0002_0018.ENC_Status_compact.Status/TxPDO_Toggle <-> ENC Status compact/Status/TxPDO Toggle
//     PlcTask Inputs/GVL_iXlinker.EtherCAT_Master_ERxxxx.Beckhoff_ER5xxx.Beckhoff_ER5xxxEK1122.A_0003_ER5151_0002_0018.ENC_Status_compact.Counter_value <-> ENC Status compact/Counter value
//     PlcTask Inputs/GVL_iXlinker.EtherCAT_Master_ERxxxx.Beckhoff_ER5xxx.Beckhoff_ER5xxxEK1122.A_0003_ER5151_0002_0018.ENC_Status_compact.Latch_value <-> ENC Status compact/Latch value
//     PlcTask Outputs/GVL_iXlinker.EtherCAT_Master_ERxxxx.Beckhoff_ER5xxx.Beckhoff_ER5xxxEK1122.A_0003_ER5151_0002_0018.ENC_Control_compact.Control/Enable_latch_C <-> ENC Control compact/Control/Enable latch C
//     PlcTask Outputs/GVL_iXlinker.EtherCAT_Master_ERxxxx.Beckhoff_ER5xxx.Beckhoff_ER5xxxEK1122.A_0003_ER5151_0002_0018.ENC_Control_compact.Control/Enable_latch_extern_on_positive_edge <-> ENC Control compact/Control/Enable latch extern on positive edge
//     PlcTask Outputs/GVL_iXlinker.EtherCAT_Master_ERxxxx.Beckhoff_ER5xxx.Beckhoff_ER5xxxEK1122.A_0003_ER5151_0002_0018.ENC_Control_compact.Control/Set_counter <-> ENC Control compact/Control/Set counter
//     PlcTask Outputs/GVL_iXlinker.EtherCAT_Master_ERxxxx.Beckhoff_ER5xxx.Beckhoff_ER5xxxEK1122.A_0003_ER5151_0002_0018.ENC_Control_compact.Control/Enable_latch_extern_on_negative_edge <-> ENC Control compact/Control/Enable latch extern on negative edge
//     PlcTask Outputs/GVL_iXlinker.EtherCAT_Master_ERxxxx.Beckhoff_ER5xxx.Beckhoff_ER5xxxEK1122.A_0003_ER5151_0002_0018.ENC_Control_compact.Set_counter_value <-> ENC Control compact/Set counter value
//     PlcTask Inputs/GVL_iXlinker.EtherCAT_Master_ERxxxx.Beckhoff_ER5xxx.Beckhoff_ER5xxxEK1122.A_0003_ER5151_0002_0018.WcState.WcState <-> WcState/WcState
//     PlcTask Inputs/GVL_iXlinker.EtherCAT_Master_ERxxxx.Beckhoff_ER5xxx.Beckhoff_ER5xxxEK1122.A_0003_ER5151_0002_0018.WcState.InputToggle <-> WcState/InputToggle
//     PlcTask Inputs/GVL_iXlinker.EtherCAT_Master_ERxxxx.Beckhoff_ER5xxx.Beckhoff_ER5xxxEK1122.A_0003_ER5151_0002_0018.InfoData.AdsAddr <-> InfoData/AdsAddr
//     PlcTask Inputs/GVL_iXlinker.EtherCAT_Master_ERxxxx.Beckhoff_ER5xxx.Beckhoff_ER5xxxEK1122.A_0003_ER5151_0002_0018.InfoData.State <-> InfoData/State
//   PLC/PLC Instance <-> EtherCAT Master ERxxxx/Beckhoff ER6xxx
//     PlcTask Inputs/GVL_iXlinker.EtherCAT_Master_ERxxxx.Beckhoff_ER6xxx.InfoData.State <-> InfoData/State
//   PLC/PLC Instance <-> EtherCAT Master ERxxxx/Beckhoff ER6xxx/Beckhoff ER6xxxEK1122
//     PlcTask Inputs/GVL_iXlinker.EtherCAT_Master_ERxxxx.Beckhoff_ER6xxx.Beckhoff_ER6xxxEK1122.InfoData.State <-> InfoData/State
//   PLC/PLC Instance <-> EtherCAT Master ERxxxx/Beckhoff ER6xxx/Beckhoff ER6xxxEK1122/Beckhoff ER6xxxsub EK1100
//     PlcTask Inputs/GVL_iXlinker.EtherCAT_Master_ERxxxx.Beckhoff_ER6xxx.Beckhoff_ER6xxxEK1122.Beckhoff_ER6xxxsub_EK1100.InfoData.State <-> InfoData/State
//   PLC/PLC Instance <-> EtherCAT Master ERxxxx/Beckhoff ER6xxx/Beckhoff ER6xxxEK1122/A_0001(ER6001-0002-0016)
//     PlcTask Inputs/GVL_iXlinker.EtherCAT_Master_ERxxxx.Beckhoff_ER6xxx.Beckhoff_ER6xxxEK1122.A_0001_ER6001_0002_0016.COM_Inputs.Status <-> COM Inputs/Status
//     PlcTask Inputs/GVL_iXlinker.EtherCAT_Master_ERxxxx.Beckhoff_ER6xxx.Beckhoff_ER6xxxEK1122.A_0001_ER6001_0002_0016.COM_Inputs.Data_In[0] <-> COM Inputs/Data In 0
//     PlcTask Inputs/GVL_iXlinker.EtherCAT_Master_ERxxxx.Beckhoff_ER6xxx.Beckhoff_ER6xxxEK1122.A_0001_ER6001_0002_0016.COM_Inputs.Data_In[1] <-> COM Inputs/Data In 1
//     PlcTask Inputs/GVL_iXlinker.EtherCAT_Master_ERxxxx.Beckhoff_ER6xxx.Beckhoff_ER6xxxEK1122.A_0001_ER6001_0002_0016.COM_Inputs.Data_In[2] <-> COM Inputs/Data In 2
//     PlcTask Inputs/GVL_iXlinker.EtherCAT_Master_ERxxxx.Beckhoff_ER6xxx.Beckhoff_ER6xxxEK1122.A_0001_ER6001_0002_0016.COM_Inputs.Data_In[3] <-> COM Inputs/Data In 3
//     PlcTask Inputs/GVL_iXlinker.EtherCAT_Master_ERxxxx.Beckhoff_ER6xxx.Beckhoff_ER6xxxEK1122.A_0001_ER6001_0002_0016.COM_Inputs.Data_In[4] <-> COM Inputs/Data In 4
//     PlcTask Inputs/GVL_iXlinker.EtherCAT_Master_ERxxxx.Beckhoff_ER6xxx.Beckhoff_ER6xxxEK1122.A_0001_ER6001_0002_0016.COM_Inputs.Data_In[5] <-> COM Inputs/Data In 5
//     PlcTask Inputs/GVL_iXlinker.EtherCAT_Master_ERxxxx.Beckhoff_ER6xxx.Beckhoff_ER6xxxEK1122.A_0001_ER6001_0002_0016.COM_Inputs.Data_In[6] <-> COM Inputs/Data In 6
//     PlcTask Inputs/GVL_iXlinker.EtherCAT_Master_ERxxxx.Beckhoff_ER6xxx.Beckhoff_ER6xxxEK1122.A_0001_ER6001_0002_0016.COM_Inputs.Data_In[7] <-> COM Inputs/Data In 7
//     PlcTask Inputs/GVL_iXlinker.EtherCAT_Master_ERxxxx.Beckhoff_ER6xxx.Beckhoff_ER6xxxEK1122.A_0001_ER6001_0002_0016.COM_Inputs.Data_In[8] <-> COM Inputs/Data In 8
//     PlcTask Inputs/GVL_iXlinker.EtherCAT_Master_ERxxxx.Beckhoff_ER6xxx.Beckhoff_ER6xxxEK1122.A_0001_ER6001_0002_0016.COM_Inputs.Data_In[9] <-> COM Inputs/Data In 9
//     PlcTask Inputs/GVL_iXlinker.EtherCAT_Master_ERxxxx.Beckhoff_ER6xxx.Beckhoff_ER6xxxEK1122.A_0001_ER6001_0002_0016.COM_Inputs.Data_In[10] <-> COM Inputs/Data In 10
//     PlcTask Inputs/GVL_iXlinker.EtherCAT_Master_ERxxxx.Beckhoff_ER6xxx.Beckhoff_ER6xxxEK1122.A_0001_ER6001_0002_0016.COM_Inputs.Data_In[11] <-> COM Inputs/Data In 11
//     PlcTask Inputs/GVL_iXlinker.EtherCAT_Master_ERxxxx.Beckhoff_ER6xxx.Beckhoff_ER6xxxEK1122.A_0001_ER6001_0002_0016.COM_Inputs.Data_In[12] <-> COM Inputs/Data In 12
//     PlcTask Inputs/GVL_iXlinker.EtherCAT_Master_ERxxxx.Beckhoff_ER6xxx.Beckhoff_ER6xxxEK1122.A_0001_ER6001_0002_0016.COM_Inputs.Data_In[13] <-> COM Inputs/Data In 13
//     PlcTask Inputs/GVL_iXlinker.EtherCAT_Master_ERxxxx.Beckhoff_ER6xxx.Beckhoff_ER6xxxEK1122.A_0001_ER6001_0002_0016.COM_Inputs.Data_In[14] <-> COM Inputs/Data In 14
//     PlcTask Inputs/GVL_iXlinker.EtherCAT_Master_ERxxxx.Beckhoff_ER6xxx.Beckhoff_ER6xxxEK1122.A_0001_ER6001_0002_0016.COM_Inputs.Data_In[15] <-> COM Inputs/Data In 15
//     PlcTask Inputs/GVL_iXlinker.EtherCAT_Master_ERxxxx.Beckhoff_ER6xxx.Beckhoff_ER6xxxEK1122.A_0001_ER6001_0002_0016.COM_Inputs.Data_In[16] <-> COM Inputs/Data In 16
//     PlcTask Inputs/GVL_iXlinker.EtherCAT_Master_ERxxxx.Beckhoff_ER6xxx.Beckhoff_ER6xxxEK1122.A_0001_ER6001_0002_0016.COM_Inputs.Data_In[17] <-> COM Inputs/Data In 17
//     PlcTask Inputs/GVL_iXlinker.EtherCAT_Master_ERxxxx.Beckhoff_ER6xxx.Beckhoff_ER6xxxEK1122.A_0001_ER6001_0002_0016.COM_Inputs.Data_In[18] <-> COM Inputs/Data In 18
//     PlcTask Inputs/GVL_iXlinker.EtherCAT_Master_ERxxxx.Beckhoff_ER6xxx.Beckhoff_ER6xxxEK1122.A_0001_ER6001_0002_0016.COM_Inputs.Data_In[19] <-> COM Inputs/Data In 19
//     PlcTask Inputs/GVL_iXlinker.EtherCAT_Master_ERxxxx.Beckhoff_ER6xxx.Beckhoff_ER6xxxEK1122.A_0001_ER6001_0002_0016.COM_Inputs.Data_In[20] <-> COM Inputs/Data In 20
//     PlcTask Inputs/GVL_iXlinker.EtherCAT_Master_ERxxxx.Beckhoff_ER6xxx.Beckhoff_ER6xxxEK1122.A_0001_ER6001_0002_0016.COM_Inputs.Data_In[21] <-> COM Inputs/Data In 21
//     PlcTask Outputs/GVL_iXlinker.EtherCAT_Master_ERxxxx.Beckhoff_ER6xxx.Beckhoff_ER6xxxEK1122.A_0001_ER6001_0002_0016.COM_Outputs.Ctrl <-> COM Outputs/Ctrl
//     PlcTask Outputs/GVL_iXlinker.EtherCAT_Master_ERxxxx.Beckhoff_ER6xxx.Beckhoff_ER6xxxEK1122.A_0001_ER6001_0002_0016.COM_Outputs.Data_Out[0] <-> COM Outputs/Data Out 0
//     PlcTask Outputs/GVL_iXlinker.EtherCAT_Master_ERxxxx.Beckhoff_ER6xxx.Beckhoff_ER6xxxEK1122.A_0001_ER6001_0002_0016.COM_Outputs.Data_Out[1] <-> COM Outputs/Data Out 1
//     PlcTask Outputs/GVL_iXlinker.EtherCAT_Master_ERxxxx.Beckhoff_ER6xxx.Beckhoff_ER6xxxEK1122.A_0001_ER6001_0002_0016.COM_Outputs.Data_Out[2] <-> COM Outputs/Data Out 2
//     PlcTask Outputs/GVL_iXlinker.EtherCAT_Master_ERxxxx.Beckhoff_ER6xxx.Beckhoff_ER6xxxEK1122.A_0001_ER6001_0002_0016.COM_Outputs.Data_Out[3] <-> COM Outputs/Data Out 3
//     PlcTask Outputs/GVL_iXlinker.EtherCAT_Master_ERxxxx.Beckhoff_ER6xxx.Beckhoff_ER6xxxEK1122.A_0001_ER6001_0002_0016.COM_Outputs.Data_Out[4] <-> COM Outputs/Data Out 4
//     PlcTask Outputs/GVL_iXlinker.EtherCAT_Master_ERxxxx.Beckhoff_ER6xxx.Beckhoff_ER6xxxEK1122.A_0001_ER6001_0002_0016.COM_Outputs.Data_Out[5] <-> COM Outputs/Data Out 5
//     PlcTask Outputs/GVL_iXlinker.EtherCAT_Master_ERxxxx.Beckhoff_ER6xxx.Beckhoff_ER6xxxEK1122.A_0001_ER6001_0002_0016.COM_Outputs.Data_Out[6] <-> COM Outputs/Data Out 6
//     PlcTask Outputs/GVL_iXlinker.EtherCAT_Master_ERxxxx.Beckhoff_ER6xxx.Beckhoff_ER6xxxEK1122.A_0001_ER6001_0002_0016.COM_Outputs.Data_Out[7] <-> COM Outputs/Data Out 7
//     PlcTask Outputs/GVL_iXlinker.EtherCAT_Master_ERxxxx.Beckhoff_ER6xxx.Beckhoff_ER6xxxEK1122.A_0001_ER6001_0002_0016.COM_Outputs.Data_Out[8] <-> COM Outputs/Data Out 8
//     PlcTask Outputs/GVL_iXlinker.EtherCAT_Master_ERxxxx.Beckhoff_ER6xxx.Beckhoff_ER6xxxEK1122.A_0001_ER6001_0002_0016.COM_Outputs.Data_Out[9] <-> COM Outputs/Data Out 9
//     PlcTask Outputs/GVL_iXlinker.EtherCAT_Master_ERxxxx.Beckhoff_ER6xxx.Beckhoff_ER6xxxEK1122.A_0001_ER6001_0002_0016.COM_Outputs.Data_Out[10] <-> COM Outputs/Data Out 10
//     PlcTask Outputs/GVL_iXlinker.EtherCAT_Master_ERxxxx.Beckhoff_ER6xxx.Beckhoff_ER6xxxEK1122.A_0001_ER6001_0002_0016.COM_Outputs.Data_Out[11] <-> COM Outputs/Data Out 11
//     PlcTask Outputs/GVL_iXlinker.EtherCAT_Master_ERxxxx.Beckhoff_ER6xxx.Beckhoff_ER6xxxEK1122.A_0001_ER6001_0002_0016.COM_Outputs.Data_Out[12] <-> COM Outputs/Data Out 12
//     PlcTask Outputs/GVL_iXlinker.EtherCAT_Master_ERxxxx.Beckhoff_ER6xxx.Beckhoff_ER6xxxEK1122.A_0001_ER6001_0002_0016.COM_Outputs.Data_Out[13] <-> COM Outputs/Data Out 13
//     PlcTask Outputs/GVL_iXlinker.EtherCAT_Master_ERxxxx.Beckhoff_ER6xxx.Beckhoff_ER6xxxEK1122.A_0001_ER6001_0002_0016.COM_Outputs.Data_Out[14] <-> COM Outputs/Data Out 14
//     PlcTask Outputs/GVL_iXlinker.EtherCAT_Master_ERxxxx.Beckhoff_ER6xxx.Beckhoff_ER6xxxEK1122.A_0001_ER6001_0002_0016.COM_Outputs.Data_Out[15] <-> COM Outputs/Data Out 15
//     PlcTask Outputs/GVL_iXlinker.EtherCAT_Master_ERxxxx.Beckhoff_ER6xxx.Beckhoff_ER6xxxEK1122.A_0001_ER6001_0002_0016.COM_Outputs.Data_Out[16] <-> COM Outputs/Data Out 16
//     PlcTask Outputs/GVL_iXlinker.EtherCAT_Master_ERxxxx.Beckhoff_ER6xxx.Beckhoff_ER6xxxEK1122.A_0001_ER6001_0002_0016.COM_Outputs.Data_Out[17] <-> COM Outputs/Data Out 17
//     PlcTask Outputs/GVL_iXlinker.EtherCAT_Master_ERxxxx.Beckhoff_ER6xxx.Beckhoff_ER6xxxEK1122.A_0001_ER6001_0002_0016.COM_Outputs.Data_Out[18] <-> COM Outputs/Data Out 18
//     PlcTask Outputs/GVL_iXlinker.EtherCAT_Master_ERxxxx.Beckhoff_ER6xxx.Beckhoff_ER6xxxEK1122.A_0001_ER6001_0002_0016.COM_Outputs.Data_Out[19] <-> COM Outputs/Data Out 19
//     PlcTask Outputs/GVL_iXlinker.EtherCAT_Master_ERxxxx.Beckhoff_ER6xxx.Beckhoff_ER6xxxEK1122.A_0001_ER6001_0002_0016.COM_Outputs.Data_Out[20] <-> COM Outputs/Data Out 20
//     PlcTask Outputs/GVL_iXlinker.EtherCAT_Master_ERxxxx.Beckhoff_ER6xxx.Beckhoff_ER6xxxEK1122.A_0001_ER6001_0002_0016.COM_Outputs.Data_Out[21] <-> COM Outputs/Data Out 21
//     PlcTask Inputs/GVL_iXlinker.EtherCAT_Master_ERxxxx.Beckhoff_ER6xxx.Beckhoff_ER6xxxEK1122.A_0001_ER6001_0002_0016.WcState.WcState <-> WcState/WcState
//     PlcTask Inputs/GVL_iXlinker.EtherCAT_Master_ERxxxx.Beckhoff_ER6xxx.Beckhoff_ER6xxxEK1122.A_0001_ER6001_0002_0016.WcState.InputToggle <-> WcState/InputToggle
//     PlcTask Inputs/GVL_iXlinker.EtherCAT_Master_ERxxxx.Beckhoff_ER6xxx.Beckhoff_ER6xxxEK1122.A_0001_ER6001_0002_0016.InfoData.AdsAddr <-> InfoData/AdsAddr
//     PlcTask Inputs/GVL_iXlinker.EtherCAT_Master_ERxxxx.Beckhoff_ER6xxx.Beckhoff_ER6xxxEK1122.A_0001_ER6001_0002_0016.InfoData.State <-> InfoData/State
//   PLC/PLC Instance <-> EtherCAT Master ERxxxx/Beckhoff ER6xxx/Beckhoff ER6xxxEK1122/A_0002(ER6001-0002-0021)
//     PlcTask Inputs/GVL_iXlinker.EtherCAT_Master_ERxxxx.Beckhoff_ER6xxx.Beckhoff_ER6xxxEK1122.A_0002_ER6001_0002_0021.COM_Inputs.Status <-> COM Inputs/Status
//     PlcTask Inputs/GVL_iXlinker.EtherCAT_Master_ERxxxx.Beckhoff_ER6xxx.Beckhoff_ER6xxxEK1122.A_0002_ER6001_0002_0021.COM_Inputs.Data_In[0] <-> COM Inputs/Data In 0
//     PlcTask Inputs/GVL_iXlinker.EtherCAT_Master_ERxxxx.Beckhoff_ER6xxx.Beckhoff_ER6xxxEK1122.A_0002_ER6001_0002_0021.COM_Inputs.Data_In[1] <-> COM Inputs/Data In 1
//     PlcTask Inputs/GVL_iXlinker.EtherCAT_Master_ERxxxx.Beckhoff_ER6xxx.Beckhoff_ER6xxxEK1122.A_0002_ER6001_0002_0021.COM_Inputs.Data_In[2] <-> COM Inputs/Data In 2
//     PlcTask Inputs/GVL_iXlinker.EtherCAT_Master_ERxxxx.Beckhoff_ER6xxx.Beckhoff_ER6xxxEK1122.A_0002_ER6001_0002_0021.COM_Inputs.Data_In[3] <-> COM Inputs/Data In 3
//     PlcTask Inputs/GVL_iXlinker.EtherCAT_Master_ERxxxx.Beckhoff_ER6xxx.Beckhoff_ER6xxxEK1122.A_0002_ER6001_0002_0021.COM_Inputs.Data_In[4] <-> COM Inputs/Data In 4
//     PlcTask Inputs/GVL_iXlinker.EtherCAT_Master_ERxxxx.Beckhoff_ER6xxx.Beckhoff_ER6xxxEK1122.A_0002_ER6001_0002_0021.COM_Inputs.Data_In[5] <-> COM Inputs/Data In 5
//     PlcTask Inputs/GVL_iXlinker.EtherCAT_Master_ERxxxx.Beckhoff_ER6xxx.Beckhoff_ER6xxxEK1122.A_0002_ER6001_0002_0021.COM_Inputs.Data_In[6] <-> COM Inputs/Data In 6
//     PlcTask Inputs/GVL_iXlinker.EtherCAT_Master_ERxxxx.Beckhoff_ER6xxx.Beckhoff_ER6xxxEK1122.A_0002_ER6001_0002_0021.COM_Inputs.Data_In[7] <-> COM Inputs/Data In 7
//     PlcTask Inputs/GVL_iXlinker.EtherCAT_Master_ERxxxx.Beckhoff_ER6xxx.Beckhoff_ER6xxxEK1122.A_0002_ER6001_0002_0021.COM_Inputs.Data_In[8] <-> COM Inputs/Data In 8
//     PlcTask Inputs/GVL_iXlinker.EtherCAT_Master_ERxxxx.Beckhoff_ER6xxx.Beckhoff_ER6xxxEK1122.A_0002_ER6001_0002_0021.COM_Inputs.Data_In[9] <-> COM Inputs/Data In 9
//     PlcTask Inputs/GVL_iXlinker.EtherCAT_Master_ERxxxx.Beckhoff_ER6xxx.Beckhoff_ER6xxxEK1122.A_0002_ER6001_0002_0021.COM_Inputs.Data_In[10] <-> COM Inputs/Data In 10
//     PlcTask Inputs/GVL_iXlinker.EtherCAT_Master_ERxxxx.Beckhoff_ER6xxx.Beckhoff_ER6xxxEK1122.A_0002_ER6001_0002_0021.COM_Inputs.Data_In[11] <-> COM Inputs/Data In 11
//     PlcTask Inputs/GVL_iXlinker.EtherCAT_Master_ERxxxx.Beckhoff_ER6xxx.Beckhoff_ER6xxxEK1122.A_0002_ER6001_0002_0021.COM_Inputs.Data_In[12] <-> COM Inputs/Data In 12
//     PlcTask Inputs/GVL_iXlinker.EtherCAT_Master_ERxxxx.Beckhoff_ER6xxx.Beckhoff_ER6xxxEK1122.A_0002_ER6001_0002_0021.COM_Inputs.Data_In[13] <-> COM Inputs/Data In 13
//     PlcTask Inputs/GVL_iXlinker.EtherCAT_Master_ERxxxx.Beckhoff_ER6xxx.Beckhoff_ER6xxxEK1122.A_0002_ER6001_0002_0021.COM_Inputs.Data_In[14] <-> COM Inputs/Data In 14
//     PlcTask Inputs/GVL_iXlinker.EtherCAT_Master_ERxxxx.Beckhoff_ER6xxx.Beckhoff_ER6xxxEK1122.A_0002_ER6001_0002_0021.COM_Inputs.Data_In[15] <-> COM Inputs/Data In 15
//     PlcTask Inputs/GVL_iXlinker.EtherCAT_Master_ERxxxx.Beckhoff_ER6xxx.Beckhoff_ER6xxxEK1122.A_0002_ER6001_0002_0021.COM_Inputs.Data_In[16] <-> COM Inputs/Data In 16
//     PlcTask Inputs/GVL_iXlinker.EtherCAT_Master_ERxxxx.Beckhoff_ER6xxx.Beckhoff_ER6xxxEK1122.A_0002_ER6001_0002_0021.COM_Inputs.Data_In[17] <-> COM Inputs/Data In 17
//     PlcTask Inputs/GVL_iXlinker.EtherCAT_Master_ERxxxx.Beckhoff_ER6xxx.Beckhoff_ER6xxxEK1122.A_0002_ER6001_0002_0021.COM_Inputs.Data_In[18] <-> COM Inputs/Data In 18
//     PlcTask Inputs/GVL_iXlinker.EtherCAT_Master_ERxxxx.Beckhoff_ER6xxx.Beckhoff_ER6xxxEK1122.A_0002_ER6001_0002_0021.COM_Inputs.Data_In[19] <-> COM Inputs/Data In 19
//     PlcTask Inputs/GVL_iXlinker.EtherCAT_Master_ERxxxx.Beckhoff_ER6xxx.Beckhoff_ER6xxxEK1122.A_0002_ER6001_0002_0021.COM_Inputs.Data_In[20] <-> COM Inputs/Data In 20
//     PlcTask Inputs/GVL_iXlinker.EtherCAT_Master_ERxxxx.Beckhoff_ER6xxx.Beckhoff_ER6xxxEK1122.A_0002_ER6001_0002_0021.COM_Inputs.Data_In[21] <-> COM Inputs/Data In 21
//     PlcTask Outputs/GVL_iXlinker.EtherCAT_Master_ERxxxx.Beckhoff_ER6xxx.Beckhoff_ER6xxxEK1122.A_0002_ER6001_0002_0021.COM_Outputs.Ctrl <-> COM Outputs/Ctrl
//     PlcTask Outputs/GVL_iXlinker.EtherCAT_Master_ERxxxx.Beckhoff_ER6xxx.Beckhoff_ER6xxxEK1122.A_0002_ER6001_0002_0021.COM_Outputs.Data_Out[0] <-> COM Outputs/Data Out 0
//     PlcTask Outputs/GVL_iXlinker.EtherCAT_Master_ERxxxx.Beckhoff_ER6xxx.Beckhoff_ER6xxxEK1122.A_0002_ER6001_0002_0021.COM_Outputs.Data_Out[1] <-> COM Outputs/Data Out 1
//     PlcTask Outputs/GVL_iXlinker.EtherCAT_Master_ERxxxx.Beckhoff_ER6xxx.Beckhoff_ER6xxxEK1122.A_0002_ER6001_0002_0021.COM_Outputs.Data_Out[2] <-> COM Outputs/Data Out 2
//     PlcTask Outputs/GVL_iXlinker.EtherCAT_Master_ERxxxx.Beckhoff_ER6xxx.Beckhoff_ER6xxxEK1122.A_0002_ER6001_0002_0021.COM_Outputs.Data_Out[3] <-> COM Outputs/Data Out 3
//     PlcTask Outputs/GVL_iXlinker.EtherCAT_Master_ERxxxx.Beckhoff_ER6xxx.Beckhoff_ER6xxxEK1122.A_0002_ER6001_0002_0021.COM_Outputs.Data_Out[4] <-> COM Outputs/Data Out 4
//     PlcTask Outputs/GVL_iXlinker.EtherCAT_Master_ERxxxx.Beckhoff_ER6xxx.Beckhoff_ER6xxxEK1122.A_0002_ER6001_0002_0021.COM_Outputs.Data_Out[5] <-> COM Outputs/Data Out 5
//     PlcTask Outputs/GVL_iXlinker.EtherCAT_Master_ERxxxx.Beckhoff_ER6xxx.Beckhoff_ER6xxxEK1122.A_0002_ER6001_0002_0021.COM_Outputs.Data_Out[6] <-> COM Outputs/Data Out 6
//     PlcTask Outputs/GVL_iXlinker.EtherCAT_Master_ERxxxx.Beckhoff_ER6xxx.Beckhoff_ER6xxxEK1122.A_0002_ER6001_0002_0021.COM_Outputs.Data_Out[7] <-> COM Outputs/Data Out 7
//     PlcTask Outputs/GVL_iXlinker.EtherCAT_Master_ERxxxx.Beckhoff_ER6xxx.Beckhoff_ER6xxxEK1122.A_0002_ER6001_0002_0021.COM_Outputs.Data_Out[8] <-> COM Outputs/Data Out 8
//     PlcTask Outputs/GVL_iXlinker.EtherCAT_Master_ERxxxx.Beckhoff_ER6xxx.Beckhoff_ER6xxxEK1122.A_0002_ER6001_0002_0021.COM_Outputs.Data_Out[9] <-> COM Outputs/Data Out 9
//     PlcTask Outputs/GVL_iXlinker.EtherCAT_Master_ERxxxx.Beckhoff_ER6xxx.Beckhoff_ER6xxxEK1122.A_0002_ER6001_0002_0021.COM_Outputs.Data_Out[10] <-> COM Outputs/Data Out 10
//     PlcTask Outputs/GVL_iXlinker.EtherCAT_Master_ERxxxx.Beckhoff_ER6xxx.Beckhoff_ER6xxxEK1122.A_0002_ER6001_0002_0021.COM_Outputs.Data_Out[11] <-> COM Outputs/Data Out 11
//     PlcTask Outputs/GVL_iXlinker.EtherCAT_Master_ERxxxx.Beckhoff_ER6xxx.Beckhoff_ER6xxxEK1122.A_0002_ER6001_0002_0021.COM_Outputs.Data_Out[12] <-> COM Outputs/Data Out 12
//     PlcTask Outputs/GVL_iXlinker.EtherCAT_Master_ERxxxx.Beckhoff_ER6xxx.Beckhoff_ER6xxxEK1122.A_0002_ER6001_0002_0021.COM_Outputs.Data_Out[13] <-> COM Outputs/Data Out 13
//     PlcTask Outputs/GVL_iXlinker.EtherCAT_Master_ERxxxx.Beckhoff_ER6xxx.Beckhoff_ER6xxxEK1122.A_0002_ER6001_0002_0021.COM_Outputs.Data_Out[14] <-> COM Outputs/Data Out 14
//     PlcTask Outputs/GVL_iXlinker.EtherCAT_Master_ERxxxx.Beckhoff_ER6xxx.Beckhoff_ER6xxxEK1122.A_0002_ER6001_0002_0021.COM_Outputs.Data_Out[15] <-> COM Outputs/Data Out 15
//     PlcTask Outputs/GVL_iXlinker.EtherCAT_Master_ERxxxx.Beckhoff_ER6xxx.Beckhoff_ER6xxxEK1122.A_0002_ER6001_0002_0021.COM_Outputs.Data_Out[16] <-> COM Outputs/Data Out 16
//     PlcTask Outputs/GVL_iXlinker.EtherCAT_Master_ERxxxx.Beckhoff_ER6xxx.Beckhoff_ER6xxxEK1122.A_0002_ER6001_0002_0021.COM_Outputs.Data_Out[17] <-> COM Outputs/Data Out 17
//     PlcTask Outputs/GVL_iXlinker.EtherCAT_Master_ERxxxx.Beckhoff_ER6xxx.Beckhoff_ER6xxxEK1122.A_0002_ER6001_0002_0021.COM_Outputs.Data_Out[18] <-> COM Outputs/Data Out 18
//     PlcTask Outputs/GVL_iXlinker.EtherCAT_Master_ERxxxx.Beckhoff_ER6xxx.Beckhoff_ER6xxxEK1122.A_0002_ER6001_0002_0021.COM_Outputs.Data_Out[19] <-> COM Outputs/Data Out 19
//     PlcTask Outputs/GVL_iXlinker.EtherCAT_Master_ERxxxx.Beckhoff_ER6xxx.Beckhoff_ER6xxxEK1122.A_0002_ER6001_0002_0021.COM_Outputs.Data_Out[20] <-> COM Outputs/Data Out 20
//     PlcTask Outputs/GVL_iXlinker.EtherCAT_Master_ERxxxx.Beckhoff_ER6xxx.Beckhoff_ER6xxxEK1122.A_0002_ER6001_0002_0021.COM_Outputs.Data_Out[21] <-> COM Outputs/Data Out 21
//     PlcTask Inputs/GVL_iXlinker.EtherCAT_Master_ERxxxx.Beckhoff_ER6xxx.Beckhoff_ER6xxxEK1122.A_0002_ER6001_0002_0021.WcState.WcState <-> WcState/WcState
//     PlcTask Inputs/GVL_iXlinker.EtherCAT_Master_ERxxxx.Beckhoff_ER6xxx.Beckhoff_ER6xxxEK1122.A_0002_ER6001_0002_0021.WcState.InputToggle <-> WcState/InputToggle
//     PlcTask Inputs/GVL_iXlinker.EtherCAT_Master_ERxxxx.Beckhoff_ER6xxx.Beckhoff_ER6xxxEK1122.A_0002_ER6001_0002_0021.InfoData.AdsAddr <-> InfoData/AdsAddr
//     PlcTask Inputs/GVL_iXlinker.EtherCAT_Master_ERxxxx.Beckhoff_ER6xxx.Beckhoff_ER6xxxEK1122.A_0002_ER6001_0002_0021.InfoData.State <-> InfoData/State
//   PLC/PLC Instance <-> EtherCAT Master ERxxxx/Beckhoff ER6xxx/Beckhoff ER6xxxEK1122/A_0003(ER6002-0002-0021)
//     PlcTask Inputs/GVL_iXlinker.EtherCAT_Master_ERxxxx.Beckhoff_ER6xxx.Beckhoff_ER6xxxEK1122.A_0003_ER6002_0002_0021.COM_TxPDO_Map_Inputs_Channel_1.Status <-> COM TxPDO-Map Inputs Channel 1/Status
//     PlcTask Inputs/GVL_iXlinker.EtherCAT_Master_ERxxxx.Beckhoff_ER6xxx.Beckhoff_ER6xxxEK1122.A_0003_ER6002_0002_0021.COM_TxPDO_Map_Inputs_Channel_2.Status <-> COM TxPDO-Map Inputs Channel 2/Status
//     PlcTask Inputs/GVL_iXlinker.EtherCAT_Master_ERxxxx.Beckhoff_ER6xxx.Beckhoff_ER6xxxEK1122.A_0003_ER6002_0002_0021.COM_TxPDO_Map_Inputs_Channel_1.Data_In[0] <-> COM TxPDO-Map Inputs Channel 1/Data In 0
//     PlcTask Inputs/GVL_iXlinker.EtherCAT_Master_ERxxxx.Beckhoff_ER6xxx.Beckhoff_ER6xxxEK1122.A_0003_ER6002_0002_0021.COM_TxPDO_Map_Inputs_Channel_1.Data_In[1] <-> COM TxPDO-Map Inputs Channel 1/Data In 1
//     PlcTask Inputs/GVL_iXlinker.EtherCAT_Master_ERxxxx.Beckhoff_ER6xxx.Beckhoff_ER6xxxEK1122.A_0003_ER6002_0002_0021.COM_TxPDO_Map_Inputs_Channel_1.Data_In[2] <-> COM TxPDO-Map Inputs Channel 1/Data In 2
//     PlcTask Inputs/GVL_iXlinker.EtherCAT_Master_ERxxxx.Beckhoff_ER6xxx.Beckhoff_ER6xxxEK1122.A_0003_ER6002_0002_0021.COM_TxPDO_Map_Inputs_Channel_1.Data_In[3] <-> COM TxPDO-Map Inputs Channel 1/Data In 3
//     PlcTask Inputs/GVL_iXlinker.EtherCAT_Master_ERxxxx.Beckhoff_ER6xxx.Beckhoff_ER6xxxEK1122.A_0003_ER6002_0002_0021.COM_TxPDO_Map_Inputs_Channel_1.Data_In[4] <-> COM TxPDO-Map Inputs Channel 1/Data In 4
//     PlcTask Inputs/GVL_iXlinker.EtherCAT_Master_ERxxxx.Beckhoff_ER6xxx.Beckhoff_ER6xxxEK1122.A_0003_ER6002_0002_0021.COM_TxPDO_Map_Inputs_Channel_1.Data_In[5] <-> COM TxPDO-Map Inputs Channel 1/Data In 5
//     PlcTask Inputs/GVL_iXlinker.EtherCAT_Master_ERxxxx.Beckhoff_ER6xxx.Beckhoff_ER6xxxEK1122.A_0003_ER6002_0002_0021.COM_TxPDO_Map_Inputs_Channel_1.Data_In[6] <-> COM TxPDO-Map Inputs Channel 1/Data In 6
//     PlcTask Inputs/GVL_iXlinker.EtherCAT_Master_ERxxxx.Beckhoff_ER6xxx.Beckhoff_ER6xxxEK1122.A_0003_ER6002_0002_0021.COM_TxPDO_Map_Inputs_Channel_1.Data_In[7] <-> COM TxPDO-Map Inputs Channel 1/Data In 7
//     PlcTask Inputs/GVL_iXlinker.EtherCAT_Master_ERxxxx.Beckhoff_ER6xxx.Beckhoff_ER6xxxEK1122.A_0003_ER6002_0002_0021.COM_TxPDO_Map_Inputs_Channel_1.Data_In[8] <-> COM TxPDO-Map Inputs Channel 1/Data In 8
//     PlcTask Inputs/GVL_iXlinker.EtherCAT_Master_ERxxxx.Beckhoff_ER6xxx.Beckhoff_ER6xxxEK1122.A_0003_ER6002_0002_0021.COM_TxPDO_Map_Inputs_Channel_1.Data_In[9] <-> COM TxPDO-Map Inputs Channel 1/Data In 9
//     PlcTask Inputs/GVL_iXlinker.EtherCAT_Master_ERxxxx.Beckhoff_ER6xxx.Beckhoff_ER6xxxEK1122.A_0003_ER6002_0002_0021.COM_TxPDO_Map_Inputs_Channel_1.Data_In[10] <-> COM TxPDO-Map Inputs Channel 1/Data In 10
//     PlcTask Inputs/GVL_iXlinker.EtherCAT_Master_ERxxxx.Beckhoff_ER6xxx.Beckhoff_ER6xxxEK1122.A_0003_ER6002_0002_0021.COM_TxPDO_Map_Inputs_Channel_1.Data_In[11] <-> COM TxPDO-Map Inputs Channel 1/Data In 11
//     PlcTask Inputs/GVL_iXlinker.EtherCAT_Master_ERxxxx.Beckhoff_ER6xxx.Beckhoff_ER6xxxEK1122.A_0003_ER6002_0002_0021.COM_TxPDO_Map_Inputs_Channel_1.Data_In[12] <-> COM TxPDO-Map Inputs Channel 1/Data In 12
//     PlcTask Inputs/GVL_iXlinker.EtherCAT_Master_ERxxxx.Beckhoff_ER6xxx.Beckhoff_ER6xxxEK1122.A_0003_ER6002_0002_0021.COM_TxPDO_Map_Inputs_Channel_1.Data_In[13] <-> COM TxPDO-Map Inputs Channel 1/Data In 13
//     PlcTask Inputs/GVL_iXlinker.EtherCAT_Master_ERxxxx.Beckhoff_ER6xxx.Beckhoff_ER6xxxEK1122.A_0003_ER6002_0002_0021.COM_TxPDO_Map_Inputs_Channel_1.Data_In[14] <-> COM TxPDO-Map Inputs Channel 1/Data In 14
//     PlcTask Inputs/GVL_iXlinker.EtherCAT_Master_ERxxxx.Beckhoff_ER6xxx.Beckhoff_ER6xxxEK1122.A_0003_ER6002_0002_0021.COM_TxPDO_Map_Inputs_Channel_1.Data_In[15] <-> COM TxPDO-Map Inputs Channel 1/Data In 15
//     PlcTask Inputs/GVL_iXlinker.EtherCAT_Master_ERxxxx.Beckhoff_ER6xxx.Beckhoff_ER6xxxEK1122.A_0003_ER6002_0002_0021.COM_TxPDO_Map_Inputs_Channel_1.Data_In[16] <-> COM TxPDO-Map Inputs Channel 1/Data In 16
//     PlcTask Inputs/GVL_iXlinker.EtherCAT_Master_ERxxxx.Beckhoff_ER6xxx.Beckhoff_ER6xxxEK1122.A_0003_ER6002_0002_0021.COM_TxPDO_Map_Inputs_Channel_1.Data_In[17] <-> COM TxPDO-Map Inputs Channel 1/Data In 17
//     PlcTask Inputs/GVL_iXlinker.EtherCAT_Master_ERxxxx.Beckhoff_ER6xxx.Beckhoff_ER6xxxEK1122.A_0003_ER6002_0002_0021.COM_TxPDO_Map_Inputs_Channel_1.Data_In[18] <-> COM TxPDO-Map Inputs Channel 1/Data In 18
//     PlcTask Inputs/GVL_iXlinker.EtherCAT_Master_ERxxxx.Beckhoff_ER6xxx.Beckhoff_ER6xxxEK1122.A_0003_ER6002_0002_0021.COM_TxPDO_Map_Inputs_Channel_1.Data_In[19] <-> COM TxPDO-Map Inputs Channel 1/Data In 19
//     PlcTask Inputs/GVL_iXlinker.EtherCAT_Master_ERxxxx.Beckhoff_ER6xxx.Beckhoff_ER6xxxEK1122.A_0003_ER6002_0002_0021.COM_TxPDO_Map_Inputs_Channel_1.Data_In[20] <-> COM TxPDO-Map Inputs Channel 1/Data In 20
//     PlcTask Inputs/GVL_iXlinker.EtherCAT_Master_ERxxxx.Beckhoff_ER6xxx.Beckhoff_ER6xxxEK1122.A_0003_ER6002_0002_0021.COM_TxPDO_Map_Inputs_Channel_1.Data_In[21] <-> COM TxPDO-Map Inputs Channel 1/Data In 21
//     PlcTask Inputs/GVL_iXlinker.EtherCAT_Master_ERxxxx.Beckhoff_ER6xxx.Beckhoff_ER6xxxEK1122.A_0003_ER6002_0002_0021.COM_TxPDO_Map_Inputs_Channel_2.Data_In[0] <-> COM TxPDO-Map Inputs Channel 2/Data In 0
//     PlcTask Inputs/GVL_iXlinker.EtherCAT_Master_ERxxxx.Beckhoff_ER6xxx.Beckhoff_ER6xxxEK1122.A_0003_ER6002_0002_0021.COM_TxPDO_Map_Inputs_Channel_2.Data_In[1] <-> COM TxPDO-Map Inputs Channel 2/Data In 1
//     PlcTask Inputs/GVL_iXlinker.EtherCAT_Master_ERxxxx.Beckhoff_ER6xxx.Beckhoff_ER6xxxEK1122.A_0003_ER6002_0002_0021.COM_TxPDO_Map_Inputs_Channel_2.Data_In[2] <-> COM TxPDO-Map Inputs Channel 2/Data In 2
//     PlcTask Inputs/GVL_iXlinker.EtherCAT_Master_ERxxxx.Beckhoff_ER6xxx.Beckhoff_ER6xxxEK1122.A_0003_ER6002_0002_0021.COM_TxPDO_Map_Inputs_Channel_2.Data_In[3] <-> COM TxPDO-Map Inputs Channel 2/Data In 3
//     PlcTask Inputs/GVL_iXlinker.EtherCAT_Master_ERxxxx.Beckhoff_ER6xxx.Beckhoff_ER6xxxEK1122.A_0003_ER6002_0002_0021.COM_TxPDO_Map_Inputs_Channel_2.Data_In[4] <-> COM TxPDO-Map Inputs Channel 2/Data In 4
//     PlcTask Inputs/GVL_iXlinker.EtherCAT_Master_ERxxxx.Beckhoff_ER6xxx.Beckhoff_ER6xxxEK1122.A_0003_ER6002_0002_0021.COM_TxPDO_Map_Inputs_Channel_2.Data_In[5] <-> COM TxPDO-Map Inputs Channel 2/Data In 5
//     PlcTask Inputs/GVL_iXlinker.EtherCAT_Master_ERxxxx.Beckhoff_ER6xxx.Beckhoff_ER6xxxEK1122.A_0003_ER6002_0002_0021.COM_TxPDO_Map_Inputs_Channel_2.Data_In[6] <-> COM TxPDO-Map Inputs Channel 2/Data In 6
//     PlcTask Inputs/GVL_iXlinker.EtherCAT_Master_ERxxxx.Beckhoff_ER6xxx.Beckhoff_ER6xxxEK1122.A_0003_ER6002_0002_0021.COM_TxPDO_Map_Inputs_Channel_2.Data_In[7] <-> COM TxPDO-Map Inputs Channel 2/Data In 7
//     PlcTask Inputs/GVL_iXlinker.EtherCAT_Master_ERxxxx.Beckhoff_ER6xxx.Beckhoff_ER6xxxEK1122.A_0003_ER6002_0002_0021.COM_TxPDO_Map_Inputs_Channel_2.Data_In[8] <-> COM TxPDO-Map Inputs Channel 2/Data In 8
//     PlcTask Inputs/GVL_iXlinker.EtherCAT_Master_ERxxxx.Beckhoff_ER6xxx.Beckhoff_ER6xxxEK1122.A_0003_ER6002_0002_0021.COM_TxPDO_Map_Inputs_Channel_2.Data_In[9] <-> COM TxPDO-Map Inputs Channel 2/Data In 9
//     PlcTask Inputs/GVL_iXlinker.EtherCAT_Master_ERxxxx.Beckhoff_ER6xxx.Beckhoff_ER6xxxEK1122.A_0003_ER6002_0002_0021.COM_TxPDO_Map_Inputs_Channel_2.Data_In[10] <-> COM TxPDO-Map Inputs Channel 2/Data In 10
//     PlcTask Inputs/GVL_iXlinker.EtherCAT_Master_ERxxxx.Beckhoff_ER6xxx.Beckhoff_ER6xxxEK1122.A_0003_ER6002_0002_0021.COM_TxPDO_Map_Inputs_Channel_2.Data_In[11] <-> COM TxPDO-Map Inputs Channel 2/Data In 11
//     PlcTask Inputs/GVL_iXlinker.EtherCAT_Master_ERxxxx.Beckhoff_ER6xxx.Beckhoff_ER6xxxEK1122.A_0003_ER6002_0002_0021.COM_TxPDO_Map_Inputs_Channel_2.Data_In[12] <-> COM TxPDO-Map Inputs Channel 2/Data In 12
//     PlcTask Inputs/GVL_iXlinker.EtherCAT_Master_ERxxxx.Beckhoff_ER6xxx.Beckhoff_ER6xxxEK1122.A_0003_ER6002_0002_0021.COM_TxPDO_Map_Inputs_Channel_2.Data_In[13] <-> COM TxPDO-Map Inputs Channel 2/Data In 13
//     PlcTask Inputs/GVL_iXlinker.EtherCAT_Master_ERxxxx.Beckhoff_ER6xxx.Beckhoff_ER6xxxEK1122.A_0003_ER6002_0002_0021.COM_TxPDO_Map_Inputs_Channel_2.Data_In[14] <-> COM TxPDO-Map Inputs Channel 2/Data In 14
//     PlcTask Inputs/GVL_iXlinker.EtherCAT_Master_ERxxxx.Beckhoff_ER6xxx.Beckhoff_ER6xxxEK1122.A_0003_ER6002_0002_0021.COM_TxPDO_Map_Inputs_Channel_2.Data_In[15] <-> COM TxPDO-Map Inputs Channel 2/Data In 15
//     PlcTask Inputs/GVL_iXlinker.EtherCAT_Master_ERxxxx.Beckhoff_ER6xxx.Beckhoff_ER6xxxEK1122.A_0003_ER6002_0002_0021.COM_TxPDO_Map_Inputs_Channel_2.Data_In[16] <-> COM TxPDO-Map Inputs Channel 2/Data In 16
//     PlcTask Inputs/GVL_iXlinker.EtherCAT_Master_ERxxxx.Beckhoff_ER6xxx.Beckhoff_ER6xxxEK1122.A_0003_ER6002_0002_0021.COM_TxPDO_Map_Inputs_Channel_2.Data_In[17] <-> COM TxPDO-Map Inputs Channel 2/Data In 17
//     PlcTask Inputs/GVL_iXlinker.EtherCAT_Master_ERxxxx.Beckhoff_ER6xxx.Beckhoff_ER6xxxEK1122.A_0003_ER6002_0002_0021.COM_TxPDO_Map_Inputs_Channel_2.Data_In[18] <-> COM TxPDO-Map Inputs Channel 2/Data In 18
//     PlcTask Inputs/GVL_iXlinker.EtherCAT_Master_ERxxxx.Beckhoff_ER6xxx.Beckhoff_ER6xxxEK1122.A_0003_ER6002_0002_0021.COM_TxPDO_Map_Inputs_Channel_2.Data_In[19] <-> COM TxPDO-Map Inputs Channel 2/Data In 19
//     PlcTask Inputs/GVL_iXlinker.EtherCAT_Master_ERxxxx.Beckhoff_ER6xxx.Beckhoff_ER6xxxEK1122.A_0003_ER6002_0002_0021.COM_TxPDO_Map_Inputs_Channel_2.Data_In[20] <-> COM TxPDO-Map Inputs Channel 2/Data In 20
//     PlcTask Inputs/GVL_iXlinker.EtherCAT_Master_ERxxxx.Beckhoff_ER6xxx.Beckhoff_ER6xxxEK1122.A_0003_ER6002_0002_0021.COM_TxPDO_Map_Inputs_Channel_2.Data_In[21] <-> COM TxPDO-Map Inputs Channel 2/Data In 21
//     PlcTask Outputs/GVL_iXlinker.EtherCAT_Master_ERxxxx.Beckhoff_ER6xxx.Beckhoff_ER6xxxEK1122.A_0003_ER6002_0002_0021.COM_RxPDO_Map_Outputs_Channel_1.Ctrl <-> COM RxPDO-Map Outputs Channel 1/Ctrl
//     PlcTask Outputs/GVL_iXlinker.EtherCAT_Master_ERxxxx.Beckhoff_ER6xxx.Beckhoff_ER6xxxEK1122.A_0003_ER6002_0002_0021.COM_RxPDO_Map_Outputs_Channel_2.Ctrl <-> COM RxPDO-Map Outputs Channel 2/Ctrl
//     PlcTask Outputs/GVL_iXlinker.EtherCAT_Master_ERxxxx.Beckhoff_ER6xxx.Beckhoff_ER6xxxEK1122.A_0003_ER6002_0002_0021.COM_RxPDO_Map_Outputs_Channel_1.Data_Out[0] <-> COM RxPDO-Map Outputs Channel 1/Data Out 0
//     PlcTask Outputs/GVL_iXlinker.EtherCAT_Master_ERxxxx.Beckhoff_ER6xxx.Beckhoff_ER6xxxEK1122.A_0003_ER6002_0002_0021.COM_RxPDO_Map_Outputs_Channel_1.Data_Out[1] <-> COM RxPDO-Map Outputs Channel 1/Data Out 1
//     PlcTask Outputs/GVL_iXlinker.EtherCAT_Master_ERxxxx.Beckhoff_ER6xxx.Beckhoff_ER6xxxEK1122.A_0003_ER6002_0002_0021.COM_RxPDO_Map_Outputs_Channel_1.Data_Out[2] <-> COM RxPDO-Map Outputs Channel 1/Data Out 2
//     PlcTask Outputs/GVL_iXlinker.EtherCAT_Master_ERxxxx.Beckhoff_ER6xxx.Beckhoff_ER6xxxEK1122.A_0003_ER6002_0002_0021.COM_RxPDO_Map_Outputs_Channel_1.Data_Out[3] <-> COM RxPDO-Map Outputs Channel 1/Data Out 3
//     PlcTask Outputs/GVL_iXlinker.EtherCAT_Master_ERxxxx.Beckhoff_ER6xxx.Beckhoff_ER6xxxEK1122.A_0003_ER6002_0002_0021.COM_RxPDO_Map_Outputs_Channel_1.Data_Out[4] <-> COM RxPDO-Map Outputs Channel 1/Data Out 4
//     PlcTask Outputs/GVL_iXlinker.EtherCAT_Master_ERxxxx.Beckhoff_ER6xxx.Beckhoff_ER6xxxEK1122.A_0003_ER6002_0002_0021.COM_RxPDO_Map_Outputs_Channel_1.Data_Out[5] <-> COM RxPDO-Map Outputs Channel 1/Data Out 5
//     PlcTask Outputs/GVL_iXlinker.EtherCAT_Master_ERxxxx.Beckhoff_ER6xxx.Beckhoff_ER6xxxEK1122.A_0003_ER6002_0002_0021.COM_RxPDO_Map_Outputs_Channel_1.Data_Out[6] <-> COM RxPDO-Map Outputs Channel 1/Data Out 6
//     PlcTask Outputs/GVL_iXlinker.EtherCAT_Master_ERxxxx.Beckhoff_ER6xxx.Beckhoff_ER6xxxEK1122.A_0003_ER6002_0002_0021.COM_RxPDO_Map_Outputs_Channel_1.Data_Out[7] <-> COM RxPDO-Map Outputs Channel 1/Data Out 7
//     PlcTask Outputs/GVL_iXlinker.EtherCAT_Master_ERxxxx.Beckhoff_ER6xxx.Beckhoff_ER6xxxEK1122.A_0003_ER6002_0002_0021.COM_RxPDO_Map_Outputs_Channel_1.Data_Out[8] <-> COM RxPDO-Map Outputs Channel 1/Data Out 8
//     PlcTask Outputs/GVL_iXlinker.EtherCAT_Master_ERxxxx.Beckhoff_ER6xxx.Beckhoff_ER6xxxEK1122.A_0003_ER6002_0002_0021.COM_RxPDO_Map_Outputs_Channel_1.Data_Out[9] <-> COM RxPDO-Map Outputs Channel 1/Data Out 9
//     PlcTask Outputs/GVL_iXlinker.EtherCAT_Master_ERxxxx.Beckhoff_ER6xxx.Beckhoff_ER6xxxEK1122.A_0003_ER6002_0002_0021.COM_RxPDO_Map_Outputs_Channel_1.Data_Out[10] <-> COM RxPDO-Map Outputs Channel 1/Data Out 10
//     PlcTask Outputs/GVL_iXlinker.EtherCAT_Master_ERxxxx.Beckhoff_ER6xxx.Beckhoff_ER6xxxEK1122.A_0003_ER6002_0002_0021.COM_RxPDO_Map_Outputs_Channel_1.Data_Out[11] <-> COM RxPDO-Map Outputs Channel 1/Data Out 11
//     PlcTask Outputs/GVL_iXlinker.EtherCAT_Master_ERxxxx.Beckhoff_ER6xxx.Beckhoff_ER6xxxEK1122.A_0003_ER6002_0002_0021.COM_RxPDO_Map_Outputs_Channel_1.Data_Out[12] <-> COM RxPDO-Map Outputs Channel 1/Data Out 12
//     PlcTask Outputs/GVL_iXlinker.EtherCAT_Master_ERxxxx.Beckhoff_ER6xxx.Beckhoff_ER6xxxEK1122.A_0003_ER6002_0002_0021.COM_RxPDO_Map_Outputs_Channel_1.Data_Out[13] <-> COM RxPDO-Map Outputs Channel 1/Data Out 13
//     PlcTask Outputs/GVL_iXlinker.EtherCAT_Master_ERxxxx.Beckhoff_ER6xxx.Beckhoff_ER6xxxEK1122.A_0003_ER6002_0002_0021.COM_RxPDO_Map_Outputs_Channel_1.Data_Out[14] <-> COM RxPDO-Map Outputs Channel 1/Data Out 14
//     PlcTask Outputs/GVL_iXlinker.EtherCAT_Master_ERxxxx.Beckhoff_ER6xxx.Beckhoff_ER6xxxEK1122.A_0003_ER6002_0002_0021.COM_RxPDO_Map_Outputs_Channel_1.Data_Out[15] <-> COM RxPDO-Map Outputs Channel 1/Data Out 15
//     PlcTask Outputs/GVL_iXlinker.EtherCAT_Master_ERxxxx.Beckhoff_ER6xxx.Beckhoff_ER6xxxEK1122.A_0003_ER6002_0002_0021.COM_RxPDO_Map_Outputs_Channel_1.Data_Out[16] <-> COM RxPDO-Map Outputs Channel 1/Data Out 16
//     PlcTask Outputs/GVL_iXlinker.EtherCAT_Master_ERxxxx.Beckhoff_ER6xxx.Beckhoff_ER6xxxEK1122.A_0003_ER6002_0002_0021.COM_RxPDO_Map_Outputs_Channel_1.Data_Out[17] <-> COM RxPDO-Map Outputs Channel 1/Data Out 17
//     PlcTask Outputs/GVL_iXlinker.EtherCAT_Master_ERxxxx.Beckhoff_ER6xxx.Beckhoff_ER6xxxEK1122.A_0003_ER6002_0002_0021.COM_RxPDO_Map_Outputs_Channel_1.Data_Out[18] <-> COM RxPDO-Map Outputs Channel 1/Data Out 18
//     PlcTask Outputs/GVL_iXlinker.EtherCAT_Master_ERxxxx.Beckhoff_ER6xxx.Beckhoff_ER6xxxEK1122.A_0003_ER6002_0002_0021.COM_RxPDO_Map_Outputs_Channel_1.Data_Out[19] <-> COM RxPDO-Map Outputs Channel 1/Data Out 19
//     PlcTask Outputs/GVL_iXlinker.EtherCAT_Master_ERxxxx.Beckhoff_ER6xxx.Beckhoff_ER6xxxEK1122.A_0003_ER6002_0002_0021.COM_RxPDO_Map_Outputs_Channel_1.Data_Out[20] <-> COM RxPDO-Map Outputs Channel 1/Data Out 20
//     PlcTask Outputs/GVL_iXlinker.EtherCAT_Master_ERxxxx.Beckhoff_ER6xxx.Beckhoff_ER6xxxEK1122.A_0003_ER6002_0002_0021.COM_RxPDO_Map_Outputs_Channel_1.Data_Out[21] <-> COM RxPDO-Map Outputs Channel 1/Data Out 21
//     PlcTask Outputs/GVL_iXlinker.EtherCAT_Master_ERxxxx.Beckhoff_ER6xxx.Beckhoff_ER6xxxEK1122.A_0003_ER6002_0002_0021.COM_RxPDO_Map_Outputs_Channel_2.Data_Out[0] <-> COM RxPDO-Map Outputs Channel 2/Data Out 0
//     PlcTask Outputs/GVL_iXlinker.EtherCAT_Master_ERxxxx.Beckhoff_ER6xxx.Beckhoff_ER6xxxEK1122.A_0003_ER6002_0002_0021.COM_RxPDO_Map_Outputs_Channel_2.Data_Out[1] <-> COM RxPDO-Map Outputs Channel 2/Data Out 1
//     PlcTask Outputs/GVL_iXlinker.EtherCAT_Master_ERxxxx.Beckhoff_ER6xxx.Beckhoff_ER6xxxEK1122.A_0003_ER6002_0002_0021.COM_RxPDO_Map_Outputs_Channel_2.Data_Out[2] <-> COM RxPDO-Map Outputs Channel 2/Data Out 2
//     PlcTask Outputs/GVL_iXlinker.EtherCAT_Master_ERxxxx.Beckhoff_ER6xxx.Beckhoff_ER6xxxEK1122.A_0003_ER6002_0002_0021.COM_RxPDO_Map_Outputs_Channel_2.Data_Out[3] <-> COM RxPDO-Map Outputs Channel 2/Data Out 3
//     PlcTask Outputs/GVL_iXlinker.EtherCAT_Master_ERxxxx.Beckhoff_ER6xxx.Beckhoff_ER6xxxEK1122.A_0003_ER6002_0002_0021.COM_RxPDO_Map_Outputs_Channel_2.Data_Out[4] <-> COM RxPDO-Map Outputs Channel 2/Data Out 4
//     PlcTask Outputs/GVL_iXlinker.EtherCAT_Master_ERxxxx.Beckhoff_ER6xxx.Beckhoff_ER6xxxEK1122.A_0003_ER6002_0002_0021.COM_RxPDO_Map_Outputs_Channel_2.Data_Out[5] <-> COM RxPDO-Map Outputs Channel 2/Data Out 5
//     PlcTask Outputs/GVL_iXlinker.EtherCAT_Master_ERxxxx.Beckhoff_ER6xxx.Beckhoff_ER6xxxEK1122.A_0003_ER6002_0002_0021.COM_RxPDO_Map_Outputs_Channel_2.Data_Out[6] <-> COM RxPDO-Map Outputs Channel 2/Data Out 6
//     PlcTask Outputs/GVL_iXlinker.EtherCAT_Master_ERxxxx.Beckhoff_ER6xxx.Beckhoff_ER6xxxEK1122.A_0003_ER6002_0002_0021.COM_RxPDO_Map_Outputs_Channel_2.Data_Out[7] <-> COM RxPDO-Map Outputs Channel 2/Data Out 7
//     PlcTask Outputs/GVL_iXlinker.EtherCAT_Master_ERxxxx.Beckhoff_ER6xxx.Beckhoff_ER6xxxEK1122.A_0003_ER6002_0002_0021.COM_RxPDO_Map_Outputs_Channel_2.Data_Out[8] <-> COM RxPDO-Map Outputs Channel 2/Data Out 8
//     PlcTask Outputs/GVL_iXlinker.EtherCAT_Master_ERxxxx.Beckhoff_ER6xxx.Beckhoff_ER6xxxEK1122.A_0003_ER6002_0002_0021.COM_RxPDO_Map_Outputs_Channel_2.Data_Out[9] <-> COM RxPDO-Map Outputs Channel 2/Data Out 9
//     PlcTask Outputs/GVL_iXlinker.EtherCAT_Master_ERxxxx.Beckhoff_ER6xxx.Beckhoff_ER6xxxEK1122.A_0003_ER6002_0002_0021.COM_RxPDO_Map_Outputs_Channel_2.Data_Out[10] <-> COM RxPDO-Map Outputs Channel 2/Data Out 10
//     PlcTask Outputs/GVL_iXlinker.EtherCAT_Master_ERxxxx.Beckhoff_ER6xxx.Beckhoff_ER6xxxEK1122.A_0003_ER6002_0002_0021.COM_RxPDO_Map_Outputs_Channel_2.Data_Out[11] <-> COM RxPDO-Map Outputs Channel 2/Data Out 11
//     PlcTask Outputs/GVL_iXlinker.EtherCAT_Master_ERxxxx.Beckhoff_ER6xxx.Beckhoff_ER6xxxEK1122.A_0003_ER6002_0002_0021.COM_RxPDO_Map_Outputs_Channel_2.Data_Out[12] <-> COM RxPDO-Map Outputs Channel 2/Data Out 12
//     PlcTask Outputs/GVL_iXlinker.EtherCAT_Master_ERxxxx.Beckhoff_ER6xxx.Beckhoff_ER6xxxEK1122.A_0003_ER6002_0002_0021.COM_RxPDO_Map_Outputs_Channel_2.Data_Out[13] <-> COM RxPDO-Map Outputs Channel 2/Data Out 13
//     PlcTask Outputs/GVL_iXlinker.EtherCAT_Master_ERxxxx.Beckhoff_ER6xxx.Beckhoff_ER6xxxEK1122.A_0003_ER6002_0002_0021.COM_RxPDO_Map_Outputs_Channel_2.Data_Out[14] <-> COM RxPDO-Map Outputs Channel 2/Data Out 14
//     PlcTask Outputs/GVL_iXlinker.EtherCAT_Master_ERxxxx.Beckhoff_ER6xxx.Beckhoff_ER6xxxEK1122.A_0003_ER6002_0002_0021.COM_RxPDO_Map_Outputs_Channel_2.Data_Out[15] <-> COM RxPDO-Map Outputs Channel 2/Data Out 15
//     PlcTask Outputs/GVL_iXlinker.EtherCAT_Master_ERxxxx.Beckhoff_ER6xxx.Beckhoff_ER6xxxEK1122.A_0003_ER6002_0002_0021.COM_RxPDO_Map_Outputs_Channel_2.Data_Out[16] <-> COM RxPDO-Map Outputs Channel 2/Data Out 16
//     PlcTask Outputs/GVL_iXlinker.EtherCAT_Master_ERxxxx.Beckhoff_ER6xxx.Beckhoff_ER6xxxEK1122.A_0003_ER6002_0002_0021.COM_RxPDO_Map_Outputs_Channel_2.Data_Out[17] <-> COM RxPDO-Map Outputs Channel 2/Data Out 17
//     PlcTask Outputs/GVL_iXlinker.EtherCAT_Master_ERxxxx.Beckhoff_ER6xxx.Beckhoff_ER6xxxEK1122.A_0003_ER6002_0002_0021.COM_RxPDO_Map_Outputs_Channel_2.Data_Out[18] <-> COM RxPDO-Map Outputs Channel 2/Data Out 18
//     PlcTask Outputs/GVL_iXlinker.EtherCAT_Master_ERxxxx.Beckhoff_ER6xxx.Beckhoff_ER6xxxEK1122.A_0003_ER6002_0002_0021.COM_RxPDO_Map_Outputs_Channel_2.Data_Out[19] <-> COM RxPDO-Map Outputs Channel 2/Data Out 19
//     PlcTask Outputs/GVL_iXlinker.EtherCAT_Master_ERxxxx.Beckhoff_ER6xxx.Beckhoff_ER6xxxEK1122.A_0003_ER6002_0002_0021.COM_RxPDO_Map_Outputs_Channel_2.Data_Out[20] <-> COM RxPDO-Map Outputs Channel 2/Data Out 20
//     PlcTask Outputs/GVL_iXlinker.EtherCAT_Master_ERxxxx.Beckhoff_ER6xxx.Beckhoff_ER6xxxEK1122.A_0003_ER6002_0002_0021.COM_RxPDO_Map_Outputs_Channel_2.Data_Out[21] <-> COM RxPDO-Map Outputs Channel 2/Data Out 21
//     PlcTask Inputs/GVL_iXlinker.EtherCAT_Master_ERxxxx.Beckhoff_ER6xxx.Beckhoff_ER6xxxEK1122.A_0003_ER6002_0002_0021.WcState.WcState <-> WcState/WcState
//     PlcTask Inputs/GVL_iXlinker.EtherCAT_Master_ERxxxx.Beckhoff_ER6xxx.Beckhoff_ER6xxxEK1122.A_0003_ER6002_0002_0021.WcState.InputToggle <-> WcState/InputToggle
//     PlcTask Inputs/GVL_iXlinker.EtherCAT_Master_ERxxxx.Beckhoff_ER6xxx.Beckhoff_ER6xxxEK1122.A_0003_ER6002_0002_0021.InfoData.AdsAddr <-> InfoData/AdsAddr
//     PlcTask Inputs/GVL_iXlinker.EtherCAT_Master_ERxxxx.Beckhoff_ER6xxx.Beckhoff_ER6xxxEK1122.A_0003_ER6002_0002_0021.InfoData.State <-> InfoData/State
//   PLC/PLC Instance <-> EtherCAT Master ERxxxx/Beckhoff ER6xxx/Beckhoff ER6xxxEK1122/A_0004(ER6002-0002-0022)
//     PlcTask Inputs/GVL_iXlinker.EtherCAT_Master_ERxxxx.Beckhoff_ER6xxx.Beckhoff_ER6xxxEK1122.A_0004_ER6002_0002_0022.COM_TxPDO_Map_Inputs_Channel_1.Status <-> COM TxPDO-Map Inputs Channel 1/Status
//     PlcTask Inputs/GVL_iXlinker.EtherCAT_Master_ERxxxx.Beckhoff_ER6xxx.Beckhoff_ER6xxxEK1122.A_0004_ER6002_0002_0022.COM_TxPDO_Map_Inputs_Channel_2.Status <-> COM TxPDO-Map Inputs Channel 2/Status
//     PlcTask Inputs/GVL_iXlinker.EtherCAT_Master_ERxxxx.Beckhoff_ER6xxx.Beckhoff_ER6xxxEK1122.A_0004_ER6002_0002_0022.COM_TxPDO_Map_Inputs_Channel_1.Data_In[0] <-> COM TxPDO-Map Inputs Channel 1/Data In 0
//     PlcTask Inputs/GVL_iXlinker.EtherCAT_Master_ERxxxx.Beckhoff_ER6xxx.Beckhoff_ER6xxxEK1122.A_0004_ER6002_0002_0022.COM_TxPDO_Map_Inputs_Channel_1.Data_In[1] <-> COM TxPDO-Map Inputs Channel 1/Data In 1
//     PlcTask Inputs/GVL_iXlinker.EtherCAT_Master_ERxxxx.Beckhoff_ER6xxx.Beckhoff_ER6xxxEK1122.A_0004_ER6002_0002_0022.COM_TxPDO_Map_Inputs_Channel_1.Data_In[2] <-> COM TxPDO-Map Inputs Channel 1/Data In 2
//     PlcTask Inputs/GVL_iXlinker.EtherCAT_Master_ERxxxx.Beckhoff_ER6xxx.Beckhoff_ER6xxxEK1122.A_0004_ER6002_0002_0022.COM_TxPDO_Map_Inputs_Channel_1.Data_In[3] <-> COM TxPDO-Map Inputs Channel 1/Data In 3
//     PlcTask Inputs/GVL_iXlinker.EtherCAT_Master_ERxxxx.Beckhoff_ER6xxx.Beckhoff_ER6xxxEK1122.A_0004_ER6002_0002_0022.COM_TxPDO_Map_Inputs_Channel_1.Data_In[4] <-> COM TxPDO-Map Inputs Channel 1/Data In 4
//     PlcTask Inputs/GVL_iXlinker.EtherCAT_Master_ERxxxx.Beckhoff_ER6xxx.Beckhoff_ER6xxxEK1122.A_0004_ER6002_0002_0022.COM_TxPDO_Map_Inputs_Channel_1.Data_In[5] <-> COM TxPDO-Map Inputs Channel 1/Data In 5
//     PlcTask Inputs/GVL_iXlinker.EtherCAT_Master_ERxxxx.Beckhoff_ER6xxx.Beckhoff_ER6xxxEK1122.A_0004_ER6002_0002_0022.COM_TxPDO_Map_Inputs_Channel_1.Data_In[6] <-> COM TxPDO-Map Inputs Channel 1/Data In 6
//     PlcTask Inputs/GVL_iXlinker.EtherCAT_Master_ERxxxx.Beckhoff_ER6xxx.Beckhoff_ER6xxxEK1122.A_0004_ER6002_0002_0022.COM_TxPDO_Map_Inputs_Channel_1.Data_In[7] <-> COM TxPDO-Map Inputs Channel 1/Data In 7
//     PlcTask Inputs/GVL_iXlinker.EtherCAT_Master_ERxxxx.Beckhoff_ER6xxx.Beckhoff_ER6xxxEK1122.A_0004_ER6002_0002_0022.COM_TxPDO_Map_Inputs_Channel_1.Data_In[8] <-> COM TxPDO-Map Inputs Channel 1/Data In 8
//     PlcTask Inputs/GVL_iXlinker.EtherCAT_Master_ERxxxx.Beckhoff_ER6xxx.Beckhoff_ER6xxxEK1122.A_0004_ER6002_0002_0022.COM_TxPDO_Map_Inputs_Channel_1.Data_In[9] <-> COM TxPDO-Map Inputs Channel 1/Data In 9
//     PlcTask Inputs/GVL_iXlinker.EtherCAT_Master_ERxxxx.Beckhoff_ER6xxx.Beckhoff_ER6xxxEK1122.A_0004_ER6002_0002_0022.COM_TxPDO_Map_Inputs_Channel_1.Data_In[10] <-> COM TxPDO-Map Inputs Channel 1/Data In 10
//     PlcTask Inputs/GVL_iXlinker.EtherCAT_Master_ERxxxx.Beckhoff_ER6xxx.Beckhoff_ER6xxxEK1122.A_0004_ER6002_0002_0022.COM_TxPDO_Map_Inputs_Channel_1.Data_In[11] <-> COM TxPDO-Map Inputs Channel 1/Data In 11
//     PlcTask Inputs/GVL_iXlinker.EtherCAT_Master_ERxxxx.Beckhoff_ER6xxx.Beckhoff_ER6xxxEK1122.A_0004_ER6002_0002_0022.COM_TxPDO_Map_Inputs_Channel_1.Data_In[12] <-> COM TxPDO-Map Inputs Channel 1/Data In 12
//     PlcTask Inputs/GVL_iXlinker.EtherCAT_Master_ERxxxx.Beckhoff_ER6xxx.Beckhoff_ER6xxxEK1122.A_0004_ER6002_0002_0022.COM_TxPDO_Map_Inputs_Channel_1.Data_In[13] <-> COM TxPDO-Map Inputs Channel 1/Data In 13
//     PlcTask Inputs/GVL_iXlinker.EtherCAT_Master_ERxxxx.Beckhoff_ER6xxx.Beckhoff_ER6xxxEK1122.A_0004_ER6002_0002_0022.COM_TxPDO_Map_Inputs_Channel_1.Data_In[14] <-> COM TxPDO-Map Inputs Channel 1/Data In 14
//     PlcTask Inputs/GVL_iXlinker.EtherCAT_Master_ERxxxx.Beckhoff_ER6xxx.Beckhoff_ER6xxxEK1122.A_0004_ER6002_0002_0022.COM_TxPDO_Map_Inputs_Channel_1.Data_In[15] <-> COM TxPDO-Map Inputs Channel 1/Data In 15
//     PlcTask Inputs/GVL_iXlinker.EtherCAT_Master_ERxxxx.Beckhoff_ER6xxx.Beckhoff_ER6xxxEK1122.A_0004_ER6002_0002_0022.COM_TxPDO_Map_Inputs_Channel_1.Data_In[16] <-> COM TxPDO-Map Inputs Channel 1/Data In 16
//     PlcTask Inputs/GVL_iXlinker.EtherCAT_Master_ERxxxx.Beckhoff_ER6xxx.Beckhoff_ER6xxxEK1122.A_0004_ER6002_0002_0022.COM_TxPDO_Map_Inputs_Channel_1.Data_In[17] <-> COM TxPDO-Map Inputs Channel 1/Data In 17
//     PlcTask Inputs/GVL_iXlinker.EtherCAT_Master_ERxxxx.Beckhoff_ER6xxx.Beckhoff_ER6xxxEK1122.A_0004_ER6002_0002_0022.COM_TxPDO_Map_Inputs_Channel_1.Data_In[18] <-> COM TxPDO-Map Inputs Channel 1/Data In 18
//     PlcTask Inputs/GVL_iXlinker.EtherCAT_Master_ERxxxx.Beckhoff_ER6xxx.Beckhoff_ER6xxxEK1122.A_0004_ER6002_0002_0022.COM_TxPDO_Map_Inputs_Channel_1.Data_In[19] <-> COM TxPDO-Map Inputs Channel 1/Data In 19
//     PlcTask Inputs/GVL_iXlinker.EtherCAT_Master_ERxxxx.Beckhoff_ER6xxx.Beckhoff_ER6xxxEK1122.A_0004_ER6002_0002_0022.COM_TxPDO_Map_Inputs_Channel_1.Data_In[20] <-> COM TxPDO-Map Inputs Channel 1/Data In 20
//     PlcTask Inputs/GVL_iXlinker.EtherCAT_Master_ERxxxx.Beckhoff_ER6xxx.Beckhoff_ER6xxxEK1122.A_0004_ER6002_0002_0022.COM_TxPDO_Map_Inputs_Channel_1.Data_In[21] <-> COM TxPDO-Map Inputs Channel 1/Data In 21
//     PlcTask Inputs/GVL_iXlinker.EtherCAT_Master_ERxxxx.Beckhoff_ER6xxx.Beckhoff_ER6xxxEK1122.A_0004_ER6002_0002_0022.COM_TxPDO_Map_Inputs_Channel_2.Data_In[0] <-> COM TxPDO-Map Inputs Channel 2/Data In 0
//     PlcTask Inputs/GVL_iXlinker.EtherCAT_Master_ERxxxx.Beckhoff_ER6xxx.Beckhoff_ER6xxxEK1122.A_0004_ER6002_0002_0022.COM_TxPDO_Map_Inputs_Channel_2.Data_In[1] <-> COM TxPDO-Map Inputs Channel 2/Data In 1
//     PlcTask Inputs/GVL_iXlinker.EtherCAT_Master_ERxxxx.Beckhoff_ER6xxx.Beckhoff_ER6xxxEK1122.A_0004_ER6002_0002_0022.COM_TxPDO_Map_Inputs_Channel_2.Data_In[2] <-> COM TxPDO-Map Inputs Channel 2/Data In 2
//     PlcTask Inputs/GVL_iXlinker.EtherCAT_Master_ERxxxx.Beckhoff_ER6xxx.Beckhoff_ER6xxxEK1122.A_0004_ER6002_0002_0022.COM_TxPDO_Map_Inputs_Channel_2.Data_In[3] <-> COM TxPDO-Map Inputs Channel 2/Data In 3
//     PlcTask Inputs/GVL_iXlinker.EtherCAT_Master_ERxxxx.Beckhoff_ER6xxx.Beckhoff_ER6xxxEK1122.A_0004_ER6002_0002_0022.COM_TxPDO_Map_Inputs_Channel_2.Data_In[4] <-> COM TxPDO-Map Inputs Channel 2/Data In 4
//     PlcTask Inputs/GVL_iXlinker.EtherCAT_Master_ERxxxx.Beckhoff_ER6xxx.Beckhoff_ER6xxxEK1122.A_0004_ER6002_0002_0022.COM_TxPDO_Map_Inputs_Channel_2.Data_In[5] <-> COM TxPDO-Map Inputs Channel 2/Data In 5
//     PlcTask Inputs/GVL_iXlinker.EtherCAT_Master_ERxxxx.Beckhoff_ER6xxx.Beckhoff_ER6xxxEK1122.A_0004_ER6002_0002_0022.COM_TxPDO_Map_Inputs_Channel_2.Data_In[6] <-> COM TxPDO-Map Inputs Channel 2/Data In 6
//     PlcTask Inputs/GVL_iXlinker.EtherCAT_Master_ERxxxx.Beckhoff_ER6xxx.Beckhoff_ER6xxxEK1122.A_0004_ER6002_0002_0022.COM_TxPDO_Map_Inputs_Channel_2.Data_In[7] <-> COM TxPDO-Map Inputs Channel 2/Data In 7
//     PlcTask Inputs/GVL_iXlinker.EtherCAT_Master_ERxxxx.Beckhoff_ER6xxx.Beckhoff_ER6xxxEK1122.A_0004_ER6002_0002_0022.COM_TxPDO_Map_Inputs_Channel_2.Data_In[8] <-> COM TxPDO-Map Inputs Channel 2/Data In 8
//     PlcTask Inputs/GVL_iXlinker.EtherCAT_Master_ERxxxx.Beckhoff_ER6xxx.Beckhoff_ER6xxxEK1122.A_0004_ER6002_0002_0022.COM_TxPDO_Map_Inputs_Channel_2.Data_In[9] <-> COM TxPDO-Map Inputs Channel 2/Data In 9
//     PlcTask Inputs/GVL_iXlinker.EtherCAT_Master_ERxxxx.Beckhoff_ER6xxx.Beckhoff_ER6xxxEK1122.A_0004_ER6002_0002_0022.COM_TxPDO_Map_Inputs_Channel_2.Data_In[10] <-> COM TxPDO-Map Inputs Channel 2/Data In 10
//     PlcTask Inputs/GVL_iXlinker.EtherCAT_Master_ERxxxx.Beckhoff_ER6xxx.Beckhoff_ER6xxxEK1122.A_0004_ER6002_0002_0022.COM_TxPDO_Map_Inputs_Channel_2.Data_In[11] <-> COM TxPDO-Map Inputs Channel 2/Data In 11
//     PlcTask Inputs/GVL_iXlinker.EtherCAT_Master_ERxxxx.Beckhoff_ER6xxx.Beckhoff_ER6xxxEK1122.A_0004_ER6002_0002_0022.COM_TxPDO_Map_Inputs_Channel_2.Data_In[12] <-> COM TxPDO-Map Inputs Channel 2/Data In 12
//     PlcTask Inputs/GVL_iXlinker.EtherCAT_Master_ERxxxx.Beckhoff_ER6xxx.Beckhoff_ER6xxxEK1122.A_0004_ER6002_0002_0022.COM_TxPDO_Map_Inputs_Channel_2.Data_In[13] <-> COM TxPDO-Map Inputs Channel 2/Data In 13
//     PlcTask Inputs/GVL_iXlinker.EtherCAT_Master_ERxxxx.Beckhoff_ER6xxx.Beckhoff_ER6xxxEK1122.A_0004_ER6002_0002_0022.COM_TxPDO_Map_Inputs_Channel_2.Data_In[14] <-> COM TxPDO-Map Inputs Channel 2/Data In 14
//     PlcTask Inputs/GVL_iXlinker.EtherCAT_Master_ERxxxx.Beckhoff_ER6xxx.Beckhoff_ER6xxxEK1122.A_0004_ER6002_0002_0022.COM_TxPDO_Map_Inputs_Channel_2.Data_In[15] <-> COM TxPDO-Map Inputs Channel 2/Data In 15
//     PlcTask Inputs/GVL_iXlinker.EtherCAT_Master_ERxxxx.Beckhoff_ER6xxx.Beckhoff_ER6xxxEK1122.A_0004_ER6002_0002_0022.COM_TxPDO_Map_Inputs_Channel_2.Data_In[16] <-> COM TxPDO-Map Inputs Channel 2/Data In 16
//     PlcTask Inputs/GVL_iXlinker.EtherCAT_Master_ERxxxx.Beckhoff_ER6xxx.Beckhoff_ER6xxxEK1122.A_0004_ER6002_0002_0022.COM_TxPDO_Map_Inputs_Channel_2.Data_In[17] <-> COM TxPDO-Map Inputs Channel 2/Data In 17
//     PlcTask Inputs/GVL_iXlinker.EtherCAT_Master_ERxxxx.Beckhoff_ER6xxx.Beckhoff_ER6xxxEK1122.A_0004_ER6002_0002_0022.COM_TxPDO_Map_Inputs_Channel_2.Data_In[18] <-> COM TxPDO-Map Inputs Channel 2/Data In 18
//     PlcTask Inputs/GVL_iXlinker.EtherCAT_Master_ERxxxx.Beckhoff_ER6xxx.Beckhoff_ER6xxxEK1122.A_0004_ER6002_0002_0022.COM_TxPDO_Map_Inputs_Channel_2.Data_In[19] <-> COM TxPDO-Map Inputs Channel 2/Data In 19
//     PlcTask Inputs/GVL_iXlinker.EtherCAT_Master_ERxxxx.Beckhoff_ER6xxx.Beckhoff_ER6xxxEK1122.A_0004_ER6002_0002_0022.COM_TxPDO_Map_Inputs_Channel_2.Data_In[20] <-> COM TxPDO-Map Inputs Channel 2/Data In 20
//     PlcTask Inputs/GVL_iXlinker.EtherCAT_Master_ERxxxx.Beckhoff_ER6xxx.Beckhoff_ER6xxxEK1122.A_0004_ER6002_0002_0022.COM_TxPDO_Map_Inputs_Channel_2.Data_In[21] <-> COM TxPDO-Map Inputs Channel 2/Data In 21
//     PlcTask Outputs/GVL_iXlinker.EtherCAT_Master_ERxxxx.Beckhoff_ER6xxx.Beckhoff_ER6xxxEK1122.A_0004_ER6002_0002_0022.COM_RxPDO_Map_Outputs_Channel_1.Ctrl <-> COM RxPDO-Map Outputs Channel 1/Ctrl
//     PlcTask Outputs/GVL_iXlinker.EtherCAT_Master_ERxxxx.Beckhoff_ER6xxx.Beckhoff_ER6xxxEK1122.A_0004_ER6002_0002_0022.COM_RxPDO_Map_Outputs_Channel_2.Ctrl <-> COM RxPDO-Map Outputs Channel 2/Ctrl
//     PlcTask Outputs/GVL_iXlinker.EtherCAT_Master_ERxxxx.Beckhoff_ER6xxx.Beckhoff_ER6xxxEK1122.A_0004_ER6002_0002_0022.COM_RxPDO_Map_Outputs_Channel_1.Data_Out[0] <-> COM RxPDO-Map Outputs Channel 1/Data Out 0
//     PlcTask Outputs/GVL_iXlinker.EtherCAT_Master_ERxxxx.Beckhoff_ER6xxx.Beckhoff_ER6xxxEK1122.A_0004_ER6002_0002_0022.COM_RxPDO_Map_Outputs_Channel_1.Data_Out[1] <-> COM RxPDO-Map Outputs Channel 1/Data Out 1
//     PlcTask Outputs/GVL_iXlinker.EtherCAT_Master_ERxxxx.Beckhoff_ER6xxx.Beckhoff_ER6xxxEK1122.A_0004_ER6002_0002_0022.COM_RxPDO_Map_Outputs_Channel_1.Data_Out[2] <-> COM RxPDO-Map Outputs Channel 1/Data Out 2
//     PlcTask Outputs/GVL_iXlinker.EtherCAT_Master_ERxxxx.Beckhoff_ER6xxx.Beckhoff_ER6xxxEK1122.A_0004_ER6002_0002_0022.COM_RxPDO_Map_Outputs_Channel_1.Data_Out[3] <-> COM RxPDO-Map Outputs Channel 1/Data Out 3
//     PlcTask Outputs/GVL_iXlinker.EtherCAT_Master_ERxxxx.Beckhoff_ER6xxx.Beckhoff_ER6xxxEK1122.A_0004_ER6002_0002_0022.COM_RxPDO_Map_Outputs_Channel_1.Data_Out[4] <-> COM RxPDO-Map Outputs Channel 1/Data Out 4
//     PlcTask Outputs/GVL_iXlinker.EtherCAT_Master_ERxxxx.Beckhoff_ER6xxx.Beckhoff_ER6xxxEK1122.A_0004_ER6002_0002_0022.COM_RxPDO_Map_Outputs_Channel_1.Data_Out[5] <-> COM RxPDO-Map Outputs Channel 1/Data Out 5
//     PlcTask Outputs/GVL_iXlinker.EtherCAT_Master_ERxxxx.Beckhoff_ER6xxx.Beckhoff_ER6xxxEK1122.A_0004_ER6002_0002_0022.COM_RxPDO_Map_Outputs_Channel_1.Data_Out[6] <-> COM RxPDO-Map Outputs Channel 1/Data Out 6
//     PlcTask Outputs/GVL_iXlinker.EtherCAT_Master_ERxxxx.Beckhoff_ER6xxx.Beckhoff_ER6xxxEK1122.A_0004_ER6002_0002_0022.COM_RxPDO_Map_Outputs_Channel_1.Data_Out[7] <-> COM RxPDO-Map Outputs Channel 1/Data Out 7
//     PlcTask Outputs/GVL_iXlinker.EtherCAT_Master_ERxxxx.Beckhoff_ER6xxx.Beckhoff_ER6xxxEK1122.A_0004_ER6002_0002_0022.COM_RxPDO_Map_Outputs_Channel_1.Data_Out[8] <-> COM RxPDO-Map Outputs Channel 1/Data Out 8
//     PlcTask Outputs/GVL_iXlinker.EtherCAT_Master_ERxxxx.Beckhoff_ER6xxx.Beckhoff_ER6xxxEK1122.A_0004_ER6002_0002_0022.COM_RxPDO_Map_Outputs_Channel_1.Data_Out[9] <-> COM RxPDO-Map Outputs Channel 1/Data Out 9
//     PlcTask Outputs/GVL_iXlinker.EtherCAT_Master_ERxxxx.Beckhoff_ER6xxx.Beckhoff_ER6xxxEK1122.A_0004_ER6002_0002_0022.COM_RxPDO_Map_Outputs_Channel_1.Data_Out[10] <-> COM RxPDO-Map Outputs Channel 1/Data Out 10
//     PlcTask Outputs/GVL_iXlinker.EtherCAT_Master_ERxxxx.Beckhoff_ER6xxx.Beckhoff_ER6xxxEK1122.A_0004_ER6002_0002_0022.COM_RxPDO_Map_Outputs_Channel_1.Data_Out[11] <-> COM RxPDO-Map Outputs Channel 1/Data Out 11
//     PlcTask Outputs/GVL_iXlinker.EtherCAT_Master_ERxxxx.Beckhoff_ER6xxx.Beckhoff_ER6xxxEK1122.A_0004_ER6002_0002_0022.COM_RxPDO_Map_Outputs_Channel_1.Data_Out[12] <-> COM RxPDO-Map Outputs Channel 1/Data Out 12
//     PlcTask Outputs/GVL_iXlinker.EtherCAT_Master_ERxxxx.Beckhoff_ER6xxx.Beckhoff_ER6xxxEK1122.A_0004_ER6002_0002_0022.COM_RxPDO_Map_Outputs_Channel_1.Data_Out[13] <-> COM RxPDO-Map Outputs Channel 1/Data Out 13
//     PlcTask Outputs/GVL_iXlinker.EtherCAT_Master_ERxxxx.Beckhoff_ER6xxx.Beckhoff_ER6xxxEK1122.A_0004_ER6002_0002_0022.COM_RxPDO_Map_Outputs_Channel_1.Data_Out[14] <-> COM RxPDO-Map Outputs Channel 1/Data Out 14
//     PlcTask Outputs/GVL_iXlinker.EtherCAT_Master_ERxxxx.Beckhoff_ER6xxx.Beckhoff_ER6xxxEK1122.A_0004_ER6002_0002_0022.COM_RxPDO_Map_Outputs_Channel_1.Data_Out[15] <-> COM RxPDO-Map Outputs Channel 1/Data Out 15
//     PlcTask Outputs/GVL_iXlinker.EtherCAT_Master_ERxxxx.Beckhoff_ER6xxx.Beckhoff_ER6xxxEK1122.A_0004_ER6002_0002_0022.COM_RxPDO_Map_Outputs_Channel_1.Data_Out[16] <-> COM RxPDO-Map Outputs Channel 1/Data Out 16
//     PlcTask Outputs/GVL_iXlinker.EtherCAT_Master_ERxxxx.Beckhoff_ER6xxx.Beckhoff_ER6xxxEK1122.A_0004_ER6002_0002_0022.COM_RxPDO_Map_Outputs_Channel_1.Data_Out[17] <-> COM RxPDO-Map Outputs Channel 1/Data Out 17
//     PlcTask Outputs/GVL_iXlinker.EtherCAT_Master_ERxxxx.Beckhoff_ER6xxx.Beckhoff_ER6xxxEK1122.A_0004_ER6002_0002_0022.COM_RxPDO_Map_Outputs_Channel_1.Data_Out[18] <-> COM RxPDO-Map Outputs Channel 1/Data Out 18
//     PlcTask Outputs/GVL_iXlinker.EtherCAT_Master_ERxxxx.Beckhoff_ER6xxx.Beckhoff_ER6xxxEK1122.A_0004_ER6002_0002_0022.COM_RxPDO_Map_Outputs_Channel_1.Data_Out[19] <-> COM RxPDO-Map Outputs Channel 1/Data Out 19
//     PlcTask Outputs/GVL_iXlinker.EtherCAT_Master_ERxxxx.Beckhoff_ER6xxx.Beckhoff_ER6xxxEK1122.A_0004_ER6002_0002_0022.COM_RxPDO_Map_Outputs_Channel_1.Data_Out[20] <-> COM RxPDO-Map Outputs Channel 1/Data Out 20
//     PlcTask Outputs/GVL_iXlinker.EtherCAT_Master_ERxxxx.Beckhoff_ER6xxx.Beckhoff_ER6xxxEK1122.A_0004_ER6002_0002_0022.COM_RxPDO_Map_Outputs_Channel_1.Data_Out[21] <-> COM RxPDO-Map Outputs Channel 1/Data Out 21
//     PlcTask Outputs/GVL_iXlinker.EtherCAT_Master_ERxxxx.Beckhoff_ER6xxx.Beckhoff_ER6xxxEK1122.A_0004_ER6002_0002_0022.COM_RxPDO_Map_Outputs_Channel_2.Data_Out[0] <-> COM RxPDO-Map Outputs Channel 2/Data Out 0
//     PlcTask Outputs/GVL_iXlinker.EtherCAT_Master_ERxxxx.Beckhoff_ER6xxx.Beckhoff_ER6xxxEK1122.A_0004_ER6002_0002_0022.COM_RxPDO_Map_Outputs_Channel_2.Data_Out[1] <-> COM RxPDO-Map Outputs Channel 2/Data Out 1
//     PlcTask Outputs/GVL_iXlinker.EtherCAT_Master_ERxxxx.Beckhoff_ER6xxx.Beckhoff_ER6xxxEK1122.A_0004_ER6002_0002_0022.COM_RxPDO_Map_Outputs_Channel_2.Data_Out[2] <-> COM RxPDO-Map Outputs Channel 2/Data Out 2
//     PlcTask Outputs/GVL_iXlinker.EtherCAT_Master_ERxxxx.Beckhoff_ER6xxx.Beckhoff_ER6xxxEK1122.A_0004_ER6002_0002_0022.COM_RxPDO_Map_Outputs_Channel_2.Data_Out[3] <-> COM RxPDO-Map Outputs Channel 2/Data Out 3
//     PlcTask Outputs/GVL_iXlinker.EtherCAT_Master_ERxxxx.Beckhoff_ER6xxx.Beckhoff_ER6xxxEK1122.A_0004_ER6002_0002_0022.COM_RxPDO_Map_Outputs_Channel_2.Data_Out[4] <-> COM RxPDO-Map Outputs Channel 2/Data Out 4
//     PlcTask Outputs/GVL_iXlinker.EtherCAT_Master_ERxxxx.Beckhoff_ER6xxx.Beckhoff_ER6xxxEK1122.A_0004_ER6002_0002_0022.COM_RxPDO_Map_Outputs_Channel_2.Data_Out[5] <-> COM RxPDO-Map Outputs Channel 2/Data Out 5
//     PlcTask Outputs/GVL_iXlinker.EtherCAT_Master_ERxxxx.Beckhoff_ER6xxx.Beckhoff_ER6xxxEK1122.A_0004_ER6002_0002_0022.COM_RxPDO_Map_Outputs_Channel_2.Data_Out[6] <-> COM RxPDO-Map Outputs Channel 2/Data Out 6
//     PlcTask Outputs/GVL_iXlinker.EtherCAT_Master_ERxxxx.Beckhoff_ER6xxx.Beckhoff_ER6xxxEK1122.A_0004_ER6002_0002_0022.COM_RxPDO_Map_Outputs_Channel_2.Data_Out[7] <-> COM RxPDO-Map Outputs Channel 2/Data Out 7
//     PlcTask Outputs/GVL_iXlinker.EtherCAT_Master_ERxxxx.Beckhoff_ER6xxx.Beckhoff_ER6xxxEK1122.A_0004_ER6002_0002_0022.COM_RxPDO_Map_Outputs_Channel_2.Data_Out[8] <-> COM RxPDO-Map Outputs Channel 2/Data Out 8
//     PlcTask Outputs/GVL_iXlinker.EtherCAT_Master_ERxxxx.Beckhoff_ER6xxx.Beckhoff_ER6xxxEK1122.A_0004_ER6002_0002_0022.COM_RxPDO_Map_Outputs_Channel_2.Data_Out[9] <-> COM RxPDO-Map Outputs Channel 2/Data Out 9
//     PlcTask Outputs/GVL_iXlinker.EtherCAT_Master_ERxxxx.Beckhoff_ER6xxx.Beckhoff_ER6xxxEK1122.A_0004_ER6002_0002_0022.COM_RxPDO_Map_Outputs_Channel_2.Data_Out[10] <-> COM RxPDO-Map Outputs Channel 2/Data Out 10
//     PlcTask Outputs/GVL_iXlinker.EtherCAT_Master_ERxxxx.Beckhoff_ER6xxx.Beckhoff_ER6xxxEK1122.A_0004_ER6002_0002_0022.COM_RxPDO_Map_Outputs_Channel_2.Data_Out[11] <-> COM RxPDO-Map Outputs Channel 2/Data Out 11
//     PlcTask Outputs/GVL_iXlinker.EtherCAT_Master_ERxxxx.Beckhoff_ER6xxx.Beckhoff_ER6xxxEK1122.A_0004_ER6002_0002_0022.COM_RxPDO_Map_Outputs_Channel_2.Data_Out[12] <-> COM RxPDO-Map Outputs Channel 2/Data Out 12
//     PlcTask Outputs/GVL_iXlinker.EtherCAT_Master_ERxxxx.Beckhoff_ER6xxx.Beckhoff_ER6xxxEK1122.A_0004_ER6002_0002_0022.COM_RxPDO_Map_Outputs_Channel_2.Data_Out[13] <-> COM RxPDO-Map Outputs Channel 2/Data Out 13
//     PlcTask Outputs/GVL_iXlinker.EtherCAT_Master_ERxxxx.Beckhoff_ER6xxx.Beckhoff_ER6xxxEK1122.A_0004_ER6002_0002_0022.COM_RxPDO_Map_Outputs_Channel_2.Data_Out[14] <-> COM RxPDO-Map Outputs Channel 2/Data Out 14
//     PlcTask Outputs/GVL_iXlinker.EtherCAT_Master_ERxxxx.Beckhoff_ER6xxx.Beckhoff_ER6xxxEK1122.A_0004_ER6002_0002_0022.COM_RxPDO_Map_Outputs_Channel_2.Data_Out[15] <-> COM RxPDO-Map Outputs Channel 2/Data Out 15
//     PlcTask Outputs/GVL_iXlinker.EtherCAT_Master_ERxxxx.Beckhoff_ER6xxx.Beckhoff_ER6xxxEK1122.A_0004_ER6002_0002_0022.COM_RxPDO_Map_Outputs_Channel_2.Data_Out[16] <-> COM RxPDO-Map Outputs Channel 2/Data Out 16
//     PlcTask Outputs/GVL_iXlinker.EtherCAT_Master_ERxxxx.Beckhoff_ER6xxx.Beckhoff_ER6xxxEK1122.A_0004_ER6002_0002_0022.COM_RxPDO_Map_Outputs_Channel_2.Data_Out[17] <-> COM RxPDO-Map Outputs Channel 2/Data Out 17
//     PlcTask Outputs/GVL_iXlinker.EtherCAT_Master_ERxxxx.Beckhoff_ER6xxx.Beckhoff_ER6xxxEK1122.A_0004_ER6002_0002_0022.COM_RxPDO_Map_Outputs_Channel_2.Data_Out[18] <-> COM RxPDO-Map Outputs Channel 2/Data Out 18
//     PlcTask Outputs/GVL_iXlinker.EtherCAT_Master_ERxxxx.Beckhoff_ER6xxx.Beckhoff_ER6xxxEK1122.A_0004_ER6002_0002_0022.COM_RxPDO_Map_Outputs_Channel_2.Data_Out[19] <-> COM RxPDO-Map Outputs Channel 2/Data Out 19
//     PlcTask Outputs/GVL_iXlinker.EtherCAT_Master_ERxxxx.Beckhoff_ER6xxx.Beckhoff_ER6xxxEK1122.A_0004_ER6002_0002_0022.COM_RxPDO_Map_Outputs_Channel_2.Data_Out[20] <-> COM RxPDO-Map Outputs Channel 2/Data Out 20
//     PlcTask Outputs/GVL_iXlinker.EtherCAT_Master_ERxxxx.Beckhoff_ER6xxx.Beckhoff_ER6xxxEK1122.A_0004_ER6002_0002_0022.COM_RxPDO_Map_Outputs_Channel_2.Data_Out[21] <-> COM RxPDO-Map Outputs Channel 2/Data Out 21
//     PlcTask Inputs/GVL_iXlinker.EtherCAT_Master_ERxxxx.Beckhoff_ER6xxx.Beckhoff_ER6xxxEK1122.A_0004_ER6002_0002_0022.WcState.WcState <-> WcState/WcState
//     PlcTask Inputs/GVL_iXlinker.EtherCAT_Master_ERxxxx.Beckhoff_ER6xxx.Beckhoff_ER6xxxEK1122.A_0004_ER6002_0002_0022.WcState.InputToggle <-> WcState/InputToggle
//     PlcTask Inputs/GVL_iXlinker.EtherCAT_Master_ERxxxx.Beckhoff_ER6xxx.Beckhoff_ER6xxxEK1122.A_0004_ER6002_0002_0022.InfoData.AdsAddr <-> InfoData/AdsAddr
//     PlcTask Inputs/GVL_iXlinker.EtherCAT_Master_ERxxxx.Beckhoff_ER6xxx.Beckhoff_ER6xxxEK1122.A_0004_ER6002_0002_0022.InfoData.State <-> InfoData/State
//   PLC/PLC Instance <-> EtherCAT Master ERxxxx/Beckhoff ER6xxx/Beckhoff ER6xxxEK1122/A_0005(ER6002-0002-0023)
//     PlcTask Inputs/GVL_iXlinker.EtherCAT_Master_ERxxxx.Beckhoff_ER6xxx.Beckhoff_ER6xxxEK1122.A_0005_ER6002_0002_0023.COM_TxPDO_Map_Inputs_Channel_1.Status <-> COM TxPDO-Map Inputs Channel 1/Status
//     PlcTask Inputs/GVL_iXlinker.EtherCAT_Master_ERxxxx.Beckhoff_ER6xxx.Beckhoff_ER6xxxEK1122.A_0005_ER6002_0002_0023.COM_TxPDO_Map_Inputs_Channel_2.Status <-> COM TxPDO-Map Inputs Channel 2/Status
//     PlcTask Inputs/GVL_iXlinker.EtherCAT_Master_ERxxxx.Beckhoff_ER6xxx.Beckhoff_ER6xxxEK1122.A_0005_ER6002_0002_0023.COM_TxPDO_Map_Inputs_Channel_1.Data_In[0] <-> COM TxPDO-Map Inputs Channel 1/Data In 0
//     PlcTask Inputs/GVL_iXlinker.EtherCAT_Master_ERxxxx.Beckhoff_ER6xxx.Beckhoff_ER6xxxEK1122.A_0005_ER6002_0002_0023.COM_TxPDO_Map_Inputs_Channel_1.Data_In[1] <-> COM TxPDO-Map Inputs Channel 1/Data In 1
//     PlcTask Inputs/GVL_iXlinker.EtherCAT_Master_ERxxxx.Beckhoff_ER6xxx.Beckhoff_ER6xxxEK1122.A_0005_ER6002_0002_0023.COM_TxPDO_Map_Inputs_Channel_1.Data_In[2] <-> COM TxPDO-Map Inputs Channel 1/Data In 2
//     PlcTask Inputs/GVL_iXlinker.EtherCAT_Master_ERxxxx.Beckhoff_ER6xxx.Beckhoff_ER6xxxEK1122.A_0005_ER6002_0002_0023.COM_TxPDO_Map_Inputs_Channel_1.Data_In[3] <-> COM TxPDO-Map Inputs Channel 1/Data In 3
//     PlcTask Inputs/GVL_iXlinker.EtherCAT_Master_ERxxxx.Beckhoff_ER6xxx.Beckhoff_ER6xxxEK1122.A_0005_ER6002_0002_0023.COM_TxPDO_Map_Inputs_Channel_1.Data_In[4] <-> COM TxPDO-Map Inputs Channel 1/Data In 4
//     PlcTask Inputs/GVL_iXlinker.EtherCAT_Master_ERxxxx.Beckhoff_ER6xxx.Beckhoff_ER6xxxEK1122.A_0005_ER6002_0002_0023.COM_TxPDO_Map_Inputs_Channel_1.Data_In[5] <-> COM TxPDO-Map Inputs Channel 1/Data In 5
//     PlcTask Inputs/GVL_iXlinker.EtherCAT_Master_ERxxxx.Beckhoff_ER6xxx.Beckhoff_ER6xxxEK1122.A_0005_ER6002_0002_0023.COM_TxPDO_Map_Inputs_Channel_1.Data_In[6] <-> COM TxPDO-Map Inputs Channel 1/Data In 6
//     PlcTask Inputs/GVL_iXlinker.EtherCAT_Master_ERxxxx.Beckhoff_ER6xxx.Beckhoff_ER6xxxEK1122.A_0005_ER6002_0002_0023.COM_TxPDO_Map_Inputs_Channel_1.Data_In[7] <-> COM TxPDO-Map Inputs Channel 1/Data In 7
//     PlcTask Inputs/GVL_iXlinker.EtherCAT_Master_ERxxxx.Beckhoff_ER6xxx.Beckhoff_ER6xxxEK1122.A_0005_ER6002_0002_0023.COM_TxPDO_Map_Inputs_Channel_1.Data_In[8] <-> COM TxPDO-Map Inputs Channel 1/Data In 8
//     PlcTask Inputs/GVL_iXlinker.EtherCAT_Master_ERxxxx.Beckhoff_ER6xxx.Beckhoff_ER6xxxEK1122.A_0005_ER6002_0002_0023.COM_TxPDO_Map_Inputs_Channel_1.Data_In[9] <-> COM TxPDO-Map Inputs Channel 1/Data In 9
//     PlcTask Inputs/GVL_iXlinker.EtherCAT_Master_ERxxxx.Beckhoff_ER6xxx.Beckhoff_ER6xxxEK1122.A_0005_ER6002_0002_0023.COM_TxPDO_Map_Inputs_Channel_1.Data_In[10] <-> COM TxPDO-Map Inputs Channel 1/Data In 10
//     PlcTask Inputs/GVL_iXlinker.EtherCAT_Master_ERxxxx.Beckhoff_ER6xxx.Beckhoff_ER6xxxEK1122.A_0005_ER6002_0002_0023.COM_TxPDO_Map_Inputs_Channel_1.Data_In[11] <-> COM TxPDO-Map Inputs Channel 1/Data In 11
//     PlcTask Inputs/GVL_iXlinker.EtherCAT_Master_ERxxxx.Beckhoff_ER6xxx.Beckhoff_ER6xxxEK1122.A_0005_ER6002_0002_0023.COM_TxPDO_Map_Inputs_Channel_1.Data_In[12] <-> COM TxPDO-Map Inputs Channel 1/Data In 12
//     PlcTask Inputs/GVL_iXlinker.EtherCAT_Master_ERxxxx.Beckhoff_ER6xxx.Beckhoff_ER6xxxEK1122.A_0005_ER6002_0002_0023.COM_TxPDO_Map_Inputs_Channel_1.Data_In[13] <-> COM TxPDO-Map Inputs Channel 1/Data In 13
//     PlcTask Inputs/GVL_iXlinker.EtherCAT_Master_ERxxxx.Beckhoff_ER6xxx.Beckhoff_ER6xxxEK1122.A_0005_ER6002_0002_0023.COM_TxPDO_Map_Inputs_Channel_1.Data_In[14] <-> COM TxPDO-Map Inputs Channel 1/Data In 14
//     PlcTask Inputs/GVL_iXlinker.EtherCAT_Master_ERxxxx.Beckhoff_ER6xxx.Beckhoff_ER6xxxEK1122.A_0005_ER6002_0002_0023.COM_TxPDO_Map_Inputs_Channel_1.Data_In[15] <-> COM TxPDO-Map Inputs Channel 1/Data In 15
//     PlcTask Inputs/GVL_iXlinker.EtherCAT_Master_ERxxxx.Beckhoff_ER6xxx.Beckhoff_ER6xxxEK1122.A_0005_ER6002_0002_0023.COM_TxPDO_Map_Inputs_Channel_1.Data_In[16] <-> COM TxPDO-Map Inputs Channel 1/Data In 16
//     PlcTask Inputs/GVL_iXlinker.EtherCAT_Master_ERxxxx.Beckhoff_ER6xxx.Beckhoff_ER6xxxEK1122.A_0005_ER6002_0002_0023.COM_TxPDO_Map_Inputs_Channel_1.Data_In[17] <-> COM TxPDO-Map Inputs Channel 1/Data In 17
//     PlcTask Inputs/GVL_iXlinker.EtherCAT_Master_ERxxxx.Beckhoff_ER6xxx.Beckhoff_ER6xxxEK1122.A_0005_ER6002_0002_0023.COM_TxPDO_Map_Inputs_Channel_1.Data_In[18] <-> COM TxPDO-Map Inputs Channel 1/Data In 18
//     PlcTask Inputs/GVL_iXlinker.EtherCAT_Master_ERxxxx.Beckhoff_ER6xxx.Beckhoff_ER6xxxEK1122.A_0005_ER6002_0002_0023.COM_TxPDO_Map_Inputs_Channel_1.Data_In[19] <-> COM TxPDO-Map Inputs Channel 1/Data In 19
//     PlcTask Inputs/GVL_iXlinker.EtherCAT_Master_ERxxxx.Beckhoff_ER6xxx.Beckhoff_ER6xxxEK1122.A_0005_ER6002_0002_0023.COM_TxPDO_Map_Inputs_Channel_1.Data_In[20] <-> COM TxPDO-Map Inputs Channel 1/Data In 20
//     PlcTask Inputs/GVL_iXlinker.EtherCAT_Master_ERxxxx.Beckhoff_ER6xxx.Beckhoff_ER6xxxEK1122.A_0005_ER6002_0002_0023.COM_TxPDO_Map_Inputs_Channel_1.Data_In[21] <-> COM TxPDO-Map Inputs Channel 1/Data In 21
//     PlcTask Inputs/GVL_iXlinker.EtherCAT_Master_ERxxxx.Beckhoff_ER6xxx.Beckhoff_ER6xxxEK1122.A_0005_ER6002_0002_0023.COM_TxPDO_Map_Inputs_Channel_2.Data_In[0] <-> COM TxPDO-Map Inputs Channel 2/Data In 0
//     PlcTask Inputs/GVL_iXlinker.EtherCAT_Master_ERxxxx.Beckhoff_ER6xxx.Beckhoff_ER6xxxEK1122.A_0005_ER6002_0002_0023.COM_TxPDO_Map_Inputs_Channel_2.Data_In[1] <-> COM TxPDO-Map Inputs Channel 2/Data In 1
//     PlcTask Inputs/GVL_iXlinker.EtherCAT_Master_ERxxxx.Beckhoff_ER6xxx.Beckhoff_ER6xxxEK1122.A_0005_ER6002_0002_0023.COM_TxPDO_Map_Inputs_Channel_2.Data_In[2] <-> COM TxPDO-Map Inputs Channel 2/Data In 2
//     PlcTask Inputs/GVL_iXlinker.EtherCAT_Master_ERxxxx.Beckhoff_ER6xxx.Beckhoff_ER6xxxEK1122.A_0005_ER6002_0002_0023.COM_TxPDO_Map_Inputs_Channel_2.Data_In[3] <-> COM TxPDO-Map Inputs Channel 2/Data In 3
//     PlcTask Inputs/GVL_iXlinker.EtherCAT_Master_ERxxxx.Beckhoff_ER6xxx.Beckhoff_ER6xxxEK1122.A_0005_ER6002_0002_0023.COM_TxPDO_Map_Inputs_Channel_2.Data_In[4] <-> COM TxPDO-Map Inputs Channel 2/Data In 4
//     PlcTask Inputs/GVL_iXlinker.EtherCAT_Master_ERxxxx.Beckhoff_ER6xxx.Beckhoff_ER6xxxEK1122.A_0005_ER6002_0002_0023.COM_TxPDO_Map_Inputs_Channel_2.Data_In[5] <-> COM TxPDO-Map Inputs Channel 2/Data In 5
//     PlcTask Inputs/GVL_iXlinker.EtherCAT_Master_ERxxxx.Beckhoff_ER6xxx.Beckhoff_ER6xxxEK1122.A_0005_ER6002_0002_0023.COM_TxPDO_Map_Inputs_Channel_2.Data_In[6] <-> COM TxPDO-Map Inputs Channel 2/Data In 6
//     PlcTask Inputs/GVL_iXlinker.EtherCAT_Master_ERxxxx.Beckhoff_ER6xxx.Beckhoff_ER6xxxEK1122.A_0005_ER6002_0002_0023.COM_TxPDO_Map_Inputs_Channel_2.Data_In[7] <-> COM TxPDO-Map Inputs Channel 2/Data In 7
//     PlcTask Inputs/GVL_iXlinker.EtherCAT_Master_ERxxxx.Beckhoff_ER6xxx.Beckhoff_ER6xxxEK1122.A_0005_ER6002_0002_0023.COM_TxPDO_Map_Inputs_Channel_2.Data_In[8] <-> COM TxPDO-Map Inputs Channel 2/Data In 8
//     PlcTask Inputs/GVL_iXlinker.EtherCAT_Master_ERxxxx.Beckhoff_ER6xxx.Beckhoff_ER6xxxEK1122.A_0005_ER6002_0002_0023.COM_TxPDO_Map_Inputs_Channel_2.Data_In[9] <-> COM TxPDO-Map Inputs Channel 2/Data In 9
//     PlcTask Inputs/GVL_iXlinker.EtherCAT_Master_ERxxxx.Beckhoff_ER6xxx.Beckhoff_ER6xxxEK1122.A_0005_ER6002_0002_0023.COM_TxPDO_Map_Inputs_Channel_2.Data_In[10] <-> COM TxPDO-Map Inputs Channel 2/Data In 10
//     PlcTask Inputs/GVL_iXlinker.EtherCAT_Master_ERxxxx.Beckhoff_ER6xxx.Beckhoff_ER6xxxEK1122.A_0005_ER6002_0002_0023.COM_TxPDO_Map_Inputs_Channel_2.Data_In[11] <-> COM TxPDO-Map Inputs Channel 2/Data In 11
